KUKA KRL program: EPS_2_251503_MH01A_A_20251120020554.src

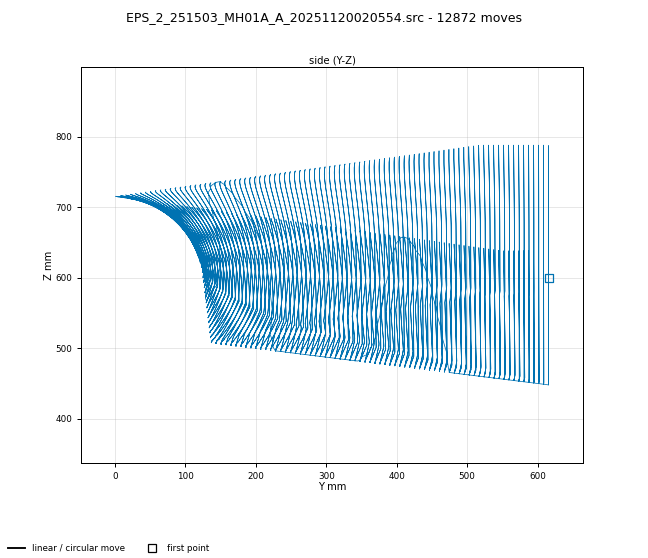
[picture p0: tool path of EPS_2_251503_MH01A_A_20251120020554.src, 12872 of 12874 moves have a stored position in this frame; points joined in program order, loops and branches not executed]
&ACCESS RVP
&REL 4
&COMMENT QRS 19112012
&PARAM EDITMASK = *
DEF PART()
EXT BAS (BAS_COMMAND :IN,REAL :IN )
INT I
BAS (#INITMOV,0 )

;KUKA QRS Post kuka4.cps  Date:22-06-2017 !

File_ID=2923

QRS_PRE_INIT()

;Init var - Until changes are made in qrs_pre_init
Outlet_Square_prg=0
Inlet_1_Square_prg=0
Inlet_2_Square_prg=0
Inlet_3_Square_prg=0
Inlet_4_Square_prg=0
Inlet_5_Square_prg=0

Outlet_1={X 0.000, Y 519.160, Z 687.500, B 0.000, E1 0.000 }
Inlet_1={X 0.000, Y 547.680, Z 287.500, B 0.000, E1 180.000 }
Outlet_1_type=201
Inlet_1_type=201
;QRS#1=Sidecore dimensions
;QRS#2=200-8" PVC SDR 35
;QRS#3=200-8" PVC SDR 35
;QRS#4=
;QRS#5=
;QRS#6=
;QRS#7=
;QRS#8=
;QRS#9=12-08 PSX
;QRS#10=12-08 PSX
;QRS#11=
;QRS#12=
;QRS#13=
;QRS#14=
;QRS#15=
;QRS#16=1220x127x1067 3,5'
;QRS#17=EPS Height
;QRS#18=788
;QRS#19=*
;QRS#20= UPDATED VERSION 22-06-2017
;QRS#21=*
Outlet_Square=0100
Inlet_1_Square=0100
Inlet_2_Square=0
Inlet_3_Square=0
Inlet_4_Square=0
Inlet_5_Square=0
Mill_Square=1
Outlet_Square_Prg=204
Inlet_1_Square_prg=204

QRS_INIT()

$ADVANCE=5

; T1
PTP {E1 173.592,E2 173.592}
PTP {X 0,Y 615.509,A -85,B 0,C 180,E1 173.592,E2 173.592,E3 0,E4 0,E5 0,E6 0}
QRS_SPEED_INIT()
LIN {X 0,Y 615.509,Z 600,A -85,B 0,C 180,E1 173.592,E2 173.592,E3 0,E4 0,E5 0,E6 0} C_VEL
LIN {X 0,Y 615.509,Z 457.87,A -85,B 0,C 180,E1 173.592,E2 173.592} C_VEL
LIN {X 0,Y 615.509,Z 449.7,A -85,B 0,C 180,E1 173.592,E2 173.592} C_VEL
LIN {X 0,Y 615.492,Z 447.7,A -85,B 0,C 180,E1 173.406,E2 173.406} C_VEL
LIN {X 0,Y 615.481,Z 447.688,A -85,B 0,C 180,E1 170.801,E2 170.801} C_VEL
LIN {X 0,Y 615.481,Z 447.684,A -85,B 0,C 180,E1 168.139,E2 168.139} C_VEL
LIN {X 0,Y 615.49,Z 447.696,A -85,B 0,C 180,E1 165.451,E2 165.451} C_VEL
LIN {X 0,Y 615.483,Z 447.687,A -85,B 0,C 180,E1 162.729,E2 162.729} C_VEL
LIN {X 0,Y 615.477,Z 447.685,A -85,B 0,C 180,E1 159.967,E2 159.967} C_VEL
LIN {X 0,Y 615.492,Z 447.699,A -85,B 0,C 180,E1 157.156,E2 157.156} C_VEL
LIN {X 0,Y 615.493,Z 447.68,A -85,B 0,C 180,E1 154.284,E2 154.284} C_VEL
LIN {X 0,Y 615.49,Z 447.696,A -85,B 0,C 180,E1 151.342,E2 151.342} C_VEL
LIN {X 0,Y 615.487,Z 447.694,A -85,B 0,C 180,E1 148.912,E2 148.912} C_VEL
LIN {X 0,Y 615.488,Z 447.684,A -85,B 0,C 180,E1 146.464,E2 146.464} C_VEL
LIN {X 0,Y 615.486,Z 447.682,A -85,B 0,C 180,E1 144.165,E2 144.165} C_VEL
LIN {X 0,Y 615.478,Z 447.684,A -85,B 0,C 180,E1 141.931,E2 141.931} C_VEL
LIN {X 0,Y 615.485,Z 447.692,A -85,B 0,C 180,E1 139.393,E2 139.393} C_VEL
LIN {X 0,Y 615.484,Z 447.693,A -85,B 0,C 180,E1 136.755,E2 136.755} C_VEL
LIN {X 0,Y 615.482,Z 447.683,A -85,B 0,C 180,E1 133.997,E2 133.997} C_VEL
LIN {X 0,Y 615.495,Z 447.698,A -85,B 0,C 180,E1 131.095,E2 131.095} C_VEL
LIN {X 0,Y 615.488,Z 447.681,A -85,B 0,C 180,E1 128.067,E2 128.067} C_VEL
LIN {X 0,Y 615.475,Z 447.687,A -85,B 0,C 180,E1 125.616,E2 125.616} C_VEL
LIN {X 0,Y 615.488,Z 447.692,A -85,B 0,C 180,E1 123.235,E2 123.235} C_VEL
LIN {X 0,Y 615.494,Z 447.701,A -85,B 0,C 180,E1 120.919,E2 120.919} C_VEL
LIN {X 0,Y 615.487,Z 447.688,A -85,B 0,C 180,E1 118.45,E2 118.45} C_VEL
LIN {X 0,Y 615.477,Z 447.684,A -85,B 0,C 180,E1 115.716,E2 115.716} C_VEL
LIN {X 0,Y 615.493,Z 447.701,A -85,B 0,C 180,E1 112.844,E2 112.844} C_VEL
LIN {X 0,Y 615.492,Z 447.681,A -85,B 0,C 180,E1 110.032,E2 110.032} C_VEL
LIN {X 0,Y 615.485,Z 447.688,A -85,B 0,C 180,E1 107.27,E2 107.27} C_VEL
LIN {X 0,Y 615.489,Z 447.693,A -85,B 0,C 180,E1 104.549,E2 104.549} C_VEL
LIN {X 0,Y 615.498,Z 447.906,A -85,B 0,C 180,E1 102.676,E2 102.676} C_VEL
LIN {X 0,Y 615.497,Z 448.814,A -85,B 0,C 180,E1 102.572,E2 102.572} C_VEL
LIN {X 0,Y 615.497,Z 534.805,A -85,B 0,C 180,E1 101.526,E2 101.526} C_VEL
LIN {X 0,Y 615.498,Z 547.747,A -85,B 0,C 180,E1 101.234,E2 101.234} C_VEL
LIN {X 0,Y 615.498,Z 560.738,A -85,B 0,C 180,E1 100.8,E2 100.8} C_VEL
LIN {X 0,Y 615.497,Z 572.199,A -85,B 0,C 180,E1 100.277,E2 100.277} C_VEL
LIN {X 0,Y 615.489,Z 583.581,A -85,B 0,C 180,E1 99.613,E2 99.613} C_VEL
LIN {X 0,Y 615.498,Z 593.825,A -85,B 0,C 180,E1 98.867,E2 98.867} C_VEL
LIN {X 0,Y 615.499,Z 603.036,A -85,B 0,C 180,E1 98.04,E2 98.04} C_VEL
LIN {X 0,Y 615.499,Z 611.893,A -85,B 0,C 180,E1 97.057,E2 97.057} C_VEL
LIN {X 0,Y 615.497,Z 619.124,A -85,B 0,C 180,E1 96.063,E2 96.063} C_VEL
LIN {X 0,Y 615.497,Z 623.959,A -85,B 0,C 180,E1 95.241,E2 95.241} C_VEL
LIN {X 0,Y 615.494,Z 628.658,A -85,B 0,C 180,E1 94.256,E2 94.256} C_VEL
LIN {X 0,Y 615.494,Z 632.255,A -85,B 0,C 180,E1 93.273,E2 93.273} C_VEL
LIN {X 0,Y 615.496,Z 634.115,A -85,B 0,C 180,E1 92.618,E2 92.618} C_VEL
LIN {X 0,Y 615.498,Z 635.533,A -85,B 0,C 180,E1 91.963,E2 91.963} C_VEL
LIN {X 0,Y 615.496,Z 637.142,A -85,B 0,C 180,E1 90.654,E2 90.654} C_VEL
LIN {X 0,Y 615.495,Z 637.384,A -85,B 0,C 180,E1 90,E2 90} C_VEL
LIN {X 0,Y 615.495,Z 637.206,A -85,B 0,C 180,E1 89.346,E2 89.346} C_VEL
LIN {X 0,Y 615.499,Z 635.682,A -85,B 0,C 180,E1 88.037,E2 88.037} C_VEL
LIN {X 0,Y 615.498,Z 634.341,A -85,B 0,C 180,E1 87.382,E2 87.382} C_VEL
LIN {X 0,Y 615.496,Z 631.494,A -85,B 0,C 180,E1 86.399,E2 86.399} C_VEL
LIN {X 0,Y 615.498,Z 627.635,A -85,B 0,C 180,E1 85.416,E2 85.416} C_VEL
LIN {X 0,Y 615.498,Z 622.652,A -85,B 0,C 180,E1 84.43,E2 84.43} C_VEL
LIN {X 0,Y 615.496,Z 616.208,A -85,B 0,C 180,E1 83.418,E2 83.418} C_VEL
LIN {X 0,Y 615.497,Z 608.538,A -85,B 0,C 180,E1 82.455,E2 82.455} C_VEL
LIN {X 0,Y 615.498,Z 598.761,A -85,B 0,C 180,E1 81.464,E2 81.464} C_VEL
LIN {X 0,Y 615.498,Z 588.496,A -85,B 0,C 180,E1 80.636,E2 80.636} C_VEL
LIN {X 0,Y 615.496,Z 576.933,A -85,B 0,C 180,E1 79.889,E2 79.889} C_VEL
LIN {X 0,Y 615.499,Z 565.025,A -85,B 0,C 180,E1 79.291,E2 79.291} C_VEL
LIN {X 0,Y 615.498,Z 552.166,A -85,B 0,C 180,E1 78.807,E2 78.807} C_VEL
LIN {X 0,Y 615.497,Z 539.569,A -85,B 0,C 180,E1 78.474,E2 78.474} C_VEL
LIN {X 0,Y 615.498,Z 526.457,A -85,B 0,C 180,E1 78.265,E2 78.265} C_VEL
LIN {X 0,Y 615.498,Z 448.939,A -85,B 0,C 180,E1 77.345,E2 77.345} C_VEL
LIN {X 0,Y 615.497,Z 447.856,A -85,B 0,C 180,E1 77.219,E2 77.219} C_VEL
LIN {X 0,Y 615.489,Z 447.691,A -85,B 0,C 180,E1 74.774,E2 74.774} C_VEL
LIN {X 0,Y 615.486,Z 447.682,A -85,B 0,C 180,E1 72.043,E2 72.043} C_VEL
LIN {X 0,Y 615.485,Z 447.696,A -85,B 0,C 180,E1 69.27,E2 69.27} C_VEL
LIN {X 0,Y 615.487,Z 447.699,A -85,B 0,C 180,E1 67.156,E2 67.156} C_VEL
LIN {X 0,Y 615.477,Z 447.687,A -85,B 0,C 180,E1 64.434,E2 64.434} C_VEL
LIN {X 0,Y 615.483,Z 447.683,A -85,B 0,C 180,E1 62.085,E2 62.085} C_VEL
LIN {X 0,Y 615.499,Z 447.679,A -85,B 0,C 180,E1 59.841,E2 59.841} C_VEL
LIN {X 0,Y 615.485,Z 447.686,A -85,B 0,C 180,E1 57.543,E2 57.543} C_VEL
LIN {X 0,Y 615.482,Z 447.696,A -85,B 0,C 180,E1 55.186,E2 55.186} C_VEL
LIN {X 0,Y 615.492,Z 447.694,A -85,B 0,C 180,E1 52.759,E2 52.759} C_VEL
LIN {X 0,Y 615.489,Z 447.681,A -85,B 0,C 180,E1 49.911,E2 49.911} C_VEL
LIN {X 0,Y 615.489,Z 447.701,A -85,B 0,C 180,E1 46.953,E2 46.953} C_VEL
LIN {X 0,Y 615.482,Z 447.683,A -85,B 0,C 180,E1 43.998,E2 43.998} C_VEL
LIN {X 0,Y 615.486,Z 447.694,A -85,B 0,C 180,E1 41.096,E2 41.096} C_VEL
LIN {X 0,Y 615.492,Z 447.7,A -85,B 0,C 180,E1 38.904,E2 38.904} C_VEL
LIN {X 0,Y 615.481,Z 447.691,A -85,B 0,C 180,E1 36.425,E2 36.425} C_VEL
LIN {X 0,Y 615.479,Z 447.684,A -85,B 0,C 180,E1 34.023,E2 34.023} C_VEL
LIN {X 0,Y 615.486,Z 447.682,A -85,B 0,C 180,E1 31.686,E2 31.686} C_VEL
LIN {X 0,Y 615.485,Z 447.685,A -85,B 0,C 180,E1 29.407,E2 29.407} C_VEL
LIN {X 0,Y 615.482,Z 447.694,A -85,B 0,C 180,E1 27.047,E2 27.047} C_VEL
LIN {X 0,Y 615.478,Z 447.69,A -85,B 0,C 180,E1 24.273,E2 24.273} C_VEL
LIN {X 0,Y 615.487,Z 447.683,A -85,B 0,C 180,E1 21.432,E2 21.432} C_VEL
LIN {X 0,Y 615.493,Z 447.698,A -85,B 0,C 180,E1 18.61,E2 18.61} C_VEL
LIN {X 0,Y 615.478,Z 447.685,A -85,B 0,C 180,E1 15.906,E2 15.906} C_VEL
LIN {X 0,Y 615.48,Z 447.687,A -85,B 0,C 180,E1 13.201,E2 13.201} C_VEL
LIN {X 0,Y 615.49,Z 447.698,A -85,B 0,C 180,E1 10.527,E2 10.527} C_VEL
LIN {X 0,Y 615.479,Z 447.685,A -85,B 0,C 180,E1 7.876,E2 7.876} C_VEL
LIN {X 0,Y 615.482,Z 447.685,A -85,B 0,C 180,E1 5.241,E2 5.241} C_VEL
LIN {X 0,Y 615.495,Z 447.699,A -85,B 0,C 180,E1 2.618,E2 2.618} C_VEL
LIN {X 0,Y 615.477,Z 447.688,A -85,B 0,C 180,E1 0,E2 0} C_VEL
LIN {X 0,Y 615.492,Z 447.681,A -85,B 0,C 180,E1 -2.618,E2 -2.618} C_VEL
LIN {X 0,Y 615.484,Z 447.695,A -85,B 0,C 180,E1 -5.241,E2 -5.241} C_VEL
LIN {X 0,Y 615.479,Z 447.692,A -85,B 0,C 180,E1 -7.876,E2 -7.876} C_VEL
LIN {X 0,Y 615.489,Z 447.681,A -85,B 0,C 180,E1 -10.527,E2 -10.527} C_VEL
LIN {X 0,Y 615.48,Z 447.693,A -85,B 0,C 180,E1 -13.201,E2 -13.201} C_VEL
LIN {X 0,Y 615.48,Z 447.693,A -85,B 0,C 180,E1 -15.905,E2 -15.905} C_VEL
LIN {X 0,Y 615.49,Z 447.681,A -85,B 0,C 180,E1 -18.646,E2 -18.646} C_VEL
LIN {X 0,Y 615.487,Z 447.696,A -85,B 0,C 180,E1 -21.432,E2 -21.432} C_VEL
LIN {X 0,Y 615.478,Z 447.686,A -85,B 0,C 180,E1 -24.272,E2 -24.272} C_VEL
LIN {X 0,Y 615.478,Z 447.687,A -85,B 0,C 180,E1 -27.046,E2 -27.046} C_VEL
LIN {X 0,Y 615.488,Z 447.698,A -85,B 0,C 180,E1 -29.797,E2 -29.797} C_VEL
LIN {X 0,Y 615.484,Z 447.683,A -85,B 0,C 180,E1 -32.458,E2 -32.458} C_VEL
LIN {X 0,Y 615.49,Z 447.681,A -85,B 0,C 180,E1 -34.815,E2 -34.815} C_VEL
LIN {X 0,Y 615.473,Z 447.69,A -85,B 0,C 180,E1 -37.243,E2 -37.243} C_VEL
LIN {X 0,Y 615.479,Z 447.693,A -85,B 0,C 180,E1 -40.09,E2 -40.09} C_VEL
LIN {X 0,Y 615.479,Z 447.687,A -85,B 0,C 180,E1 -42.354,E2 -42.354} C_VEL
LIN {X 0,Y 615.479,Z 447.685,A -85,B 0,C 180,E1 -45.07,E2 -45.07} C_VEL
LIN {X 0,Y 615.491,Z 447.698,A -85,B 0,C 180,E1 -47.92,E2 -47.92} C_VEL
LIN {X 0,Y 615.479,Z 447.69,A -85,B 0,C 180,E1 -50.25,E2 -50.25} C_VEL
LIN {X 0,Y 615.48,Z 447.684,A -85,B 0,C 180,E1 -53.065,E2 -53.065} C_VEL
LIN {X 0,Y 615.491,Z 447.698,A -85,B 0,C 180,E1 -55.979,E2 -55.979} C_VEL
LIN {X 0,Y 615.487,Z 447.682,A -85,B 0,C 180,E1 -58.914,E2 -58.914} C_VEL
LIN {X 0,Y 615.481,Z 447.692,A -85,B 0,C 180,E1 -61.551,E2 -61.551} C_VEL
LIN {X 0,Y 615.498,Z 447.813,A -85,B 0,C 180,E1 -64.013,E2 -64.013} C_VEL
LIN {X 0,Y 615.496,Z 448.16,A -85,B 0,C 180,E1 -64.104,E2 -64.104} C_VEL
LIN {X 0,Y 615.488,Z 473.307,A -85,B 0,C 180,E1 -66.801,E2 -66.801} C_VEL
LIN {X 0,Y 615.48,Z 499.798,A -85,B 0,C 180,E1 -69.577,E2 -69.577} C_VEL
LIN {X 0,Y 615.483,Z 527.091,A -85,B 0,C 180,E1 -72.387,E2 -72.387} C_VEL
LIN {X 0,Y 615.495,Z 553.944,A -85,B 0,C 180,E1 -75.113,E2 -75.113} C_VEL
LIN {X 0,Y 615.487,Z 573.871,A -85,B 0,C 180,E1 -77.093,E2 -77.093} C_VEL
LIN {X 0,Y 615.483,Z 683.847,A -85,B 0,C 180,E1 -78.411,E2 -78.411} C_VEL
LIN {X 0,Y 615.499,Z 696.352,A -85,B 0,C 180,E1 -78.682,E2 -78.682} C_VEL
LIN {X 0,Y 615.496,Z 709.5,A -85,B 0,C 180,E1 -79.109,E2 -79.109} C_VEL
LIN {X 0,Y 615.487,Z 721.482,A -85,B 0,C 180,E1 -79.64,E2 -79.64} C_VEL
LIN {X 0,Y 615.482,Z 733,A -85,B 0,C 180,E1 -80.304,E2 -80.304} C_VEL
LIN {X 0,Y 615.499,Z 743.344,A -85,B 0,C 180,E1 -81.05,E2 -81.05} C_VEL
LIN {X 0,Y 615.497,Z 751.814,A -85,B 0,C 180,E1 -81.794,E2 -81.794} C_VEL
LIN {X 0,Y 615.498,Z 759.608,A -85,B 0,C 180,E1 -82.62,E2 -82.62} C_VEL
LIN {X 0,Y 615.496,Z 767.204,A -85,B 0,C 180,E1 -83.608,E2 -83.608} C_VEL
LIN {X 0,Y 615.498,Z 774.205,A -85,B 0,C 180,E1 -84.759,E2 -84.759} C_VEL
LIN {X 0,Y 615.493,Z 778.852,A -85,B 0,C 180,E1 -85.744,E2 -85.744} C_VEL
LIN {X 0,Y 615.495,Z 782.399,A -85,B 0,C 180,E1 -86.727,E2 -86.727} C_VEL
LIN {X 0,Y 615.497,Z 784.233,A -85,B 0,C 180,E1 -87.382,E2 -87.382} C_VEL
LIN {X 0,Y 615.496,Z 785.608,A -85,B 0,C 180,E1 -88.037,E2 -88.037} C_VEL
LIN {X 0,Y 615.496,Z 787.174,A -85,B 0,C 180,E1 -89.346,E2 -89.346} C_VEL
LIN {X 0,Y 615.494,Z 787.389,A -85,B 0,C 180,E1 -90,E2 -90} C_VEL
LIN {X 0,Y 615.496,Z 786.58,A -85,B 0,C 180,E1 -91.309,E2 -91.309} C_VEL
LIN {X 0,Y 615.496,Z 785.608,A -85,B 0,C 180,E1 -91.963,E2 -91.963} C_VEL
LIN {X 0,Y 615.497,Z 784.233,A -85,B 0,C 180,E1 -92.618,E2 -92.618} C_VEL
LIN {X 0,Y 615.496,Z 781.35,A -85,B 0,C 180,E1 -93.601,E2 -93.601} C_VEL
LIN {X 0,Y 615.498,Z 777.442,A -85,B 0,C 180,E1 -94.584,E2 -94.584} C_VEL
LIN {X 0,Y 615.499,Z 772.406,A -85,B 0,C 180,E1 -95.57,E2 -95.57} C_VEL
LIN {X 0,Y 615.497,Z 765.869,A -85,B 0,C 180,E1 -96.583,E2 -96.583} C_VEL
LIN {X 0,Y 615.497,Z 758.135,A -85,B 0,C 180,E1 -97.545,E2 -97.545} C_VEL
LIN {X 0,Y 615.498,Z 750.047,A -85,B 0,C 180,E1 -98.371,E2 -98.371} C_VEL
LIN {X 0,Y 615.499,Z 740.17,A -85,B 0,C 180,E1 -99.198,E2 -99.198} C_VEL
LIN {X 0,Y 615.483,Z 728.986,A -85,B 0,C 180,E1 -99.945,E2 -99.945} C_VEL
LIN {X 0,Y 615.489,Z 718.027,A -85,B 0,C 180,E1 -100.527,E2 -100.527} C_VEL
LIN {X 0,Y 615.499,Z 705.418,A -85,B 0,C 180,E1 -101.042,E2 -101.042} C_VEL
LIN {X 0,Y 615.497,Z 693.075,A -85,B 0,C 180,E1 -101.401,E2 -101.401} C_VEL
LIN {X 0,Y 615.479,Z 679.489,A -85,B 0,C 180,E1 -101.652,E2 -101.652} C_VEL
LIN {X 0,Y 615.487,Z 573.871,A -85,B 0,C 180,E1 -102.907,E2 -102.907} C_VEL
LIN {X 0,Y 615.48,Z 548.911,A -85,B 0,C 180,E1 -105.395,E2 -105.395} C_VEL
LIN {X 0,Y 615.489,Z 522.161,A -85,B 0,C 180,E1 -108.117,E2 -108.117} C_VEL
LIN {X 0,Y 615.484,Z 495.16,A -85,B 0,C 180,E1 -110.905,E2 -110.905} C_VEL
LIN {X 0,Y 615.477,Z 468.881,A -85,B 0,C 180,E1 -113.669,E2 -113.669} C_VEL
LIN {X 0,Y 615.495,Z 448.029,A -85,B 0,C 180,E1 -115.919,E2 -115.919} C_VEL
LIN {X 0,Y 615.498,Z 447.721,A -85,B 0,C 180,E1 -116.078,E2 -116.078} C_VEL
LIN {X 0,Y 615.477,Z 447.688,A -85,B 0,C 180,E1 -118.658,E2 -118.658} C_VEL
LIN {X 0,Y 615.487,Z 447.681,A -85,B 0,C 180,E1 -121.086,E2 -121.086} C_VEL
LIN {X 0,Y 615.491,Z 447.697,A -85,B 0,C 180,E1 -124.021,E2 -124.021} C_VEL
LIN {X 0,Y 615.48,Z 447.684,A -85,B 0,C 180,E1 -126.935,E2 -126.935} C_VEL
LIN {X 0,Y 615.478,Z 447.69,A -85,B 0,C 180,E1 -129.75,E2 -129.75} C_VEL
LIN {X 0,Y 615.49,Z 447.697,A -85,B 0,C 180,E1 -132.351,E2 -132.351} C_VEL
LIN {X 0,Y 615.48,Z 447.684,A -85,B 0,C 180,E1 -135.068,E2 -135.068} C_VEL
LIN {X 0,Y 615.477,Z 447.693,A -85,B 0,C 180,E1 -137.919,E2 -137.919} C_VEL
LIN {X 0,Y 615.498,Z 447.7,A -85,B 0,C 180,E1 -140.251,E2 -140.251} C_VEL
LIN {X 0,Y 615.478,Z 447.685,A -85,B 0,C 180,E1 -143.063,E2 -143.063} C_VEL
LIN {X 0,Y 615.49,Z 447.681,A -85,B 0,C 180,E1 -145.297,E2 -145.297} C_VEL
LIN {X 0,Y 615.479,Z 447.686,A -85,B 0,C 180,E1 -147.668,E2 -147.668} C_VEL
LIN {X 0,Y 615.488,Z 447.697,A -85,B 0,C 180,E1 -150.203,E2 -150.203} C_VEL
LIN {X 0,Y 615.478,Z 447.687,A -85,B 0,C 180,E1 -152.954,E2 -152.954} C_VEL
LIN {X 0,Y 615.478,Z 447.686,A -85,B 0,C 180,E1 -155.728,E2 -155.728} C_VEL
LIN {X 0,Y 615.489,Z 447.697,A -85,B 0,C 180,E1 -158.568,E2 -158.568} C_VEL
LIN {X 0,Y 615.492,Z 447.68,A -85,B 0,C 180,E1 -161.39,E2 -161.39} C_VEL
LIN {X 0,Y 615.48,Z 447.692,A -85,B 0,C 180,E1 -164.095,E2 -164.095} C_VEL
LIN {X 0,Y 615.48,Z 447.693,A -85,B 0,C 180,E1 -166.799,E2 -166.799} C_VEL
LIN {X 0,Y 615.489,Z 447.681,A -85,B 0,C 180,E1 -169.473,E2 -169.473} C_VEL
LIN {X 0,Y 615.477,Z 447.691,A -85,B 0,C 180,E1 -172.124,E2 -172.124} C_VEL
LIN {X 0,Y 615.486,Z 447.695,A -85,B 0,C 180,E1 -174.759,E2 -174.759} C_VEL
LIN {X 0,Y 615.492,Z 447.681,A -85,B 0,C 180,E1 -177.382,E2 -177.382} C_VEL
LIN {X 0,Y 615.477,Z 447.687,A -85,B 0,C 180,E1 -180,E2 -180} C_VEL
LIN {X 0,Y 615.495,Z 447.701,A -85,B 0,C 180,E1 -182.618,E2 -182.618} C_VEL
LIN {X 0,Y 615.48,Z 447.687,A -85,B 0,C 180,E1 -185.241,E2 -185.241} C_VEL
LIN {X 0,Y 615.492,Z 447.7,A -85,B 0,C 180,E1 -186.594,E2 -186.594} C_VEL
LIN {X 0,Y 614.81,Z 447.835,A -85,B 0,C 180,E1 -187.14,E2 -187.14} C_VEL
LIN {X 0,Y 611.97,Z 448.25,A -85,B 0,C 180,E1 -188.026,E2 -188.026} C_VEL
LIN {X 0,Y 609.576,Z 448.56,A -85,B 0,C 180,E1 -188.738,E2 -188.738} C_VEL
LIN {X 0,Y 608.541,Z 448.678,A -85,B 0,C 180,E1 -189.288,E2 -189.288} C_VEL
LIN {X 0,Y 608.453,Z 448.687,A -85,B 0,C 180,E1 -189.474,E2 -189.474} C_VEL
LIN {X 0,Y 608.457,Z 448.687,A -85,B 0,C 180,E1 -192,E2 -192} C_VEL
LIN {X 0,Y 608.475,Z 448.695,A -85,B 0,C 180,E1 -194.721,E2 -194.721} C_VEL
LIN {X 0,Y 608.448,Z 448.688,A -85,B 0,C 180,E1 -197.477,E2 -197.477} C_VEL
LIN {X 0,Y 608.459,Z 448.689,A -85,B 0,C 180,E1 -200.274,E2 -200.274} C_VEL
LIN {X 0,Y 608.453,Z 448.692,A -85,B 0,C 180,E1 -203.124,E2 -203.124} C_VEL
LIN {X 0,Y 608.447,Z 448.688,A -85,B 0,C 180,E1 -206.036,E2 -206.036} C_VEL
LIN {X 0,Y 608.471,Z 448.692,A -85,B 0,C 180,E1 -208.622,E2 -208.622} C_VEL
LIN {X 0,Y 608.472,Z 448.687,A -85,B 0,C 180,E1 -211.316,E2 -211.316} C_VEL
LIN {X 0,Y 608.471,Z 448.685,A -85,B 0,C 180,E1 -213.737,E2 -213.737} C_VEL
LIN {X 0,Y 608.472,Z 448.685,A -85,B 0,C 180,E1 -216.091,E2 -216.091} C_VEL
LIN {X 0,Y 608.471,Z 448.69,A -85,B 0,C 180,E1 -218.588,E2 -218.588} C_VEL
LIN {X 0,Y 608.463,Z 448.689,A -85,B 0,C 180,E1 -221.344,E2 -221.344} C_VEL
LIN {X 0,Y 608.449,Z 448.688,A -85,B 0,C 180,E1 -224.265,E2 -224.265} C_VEL
LIN {X 0,Y 608.46,Z 448.696,A -85,B 0,C 180,E1 -227.042,E2 -227.042} C_VEL
LIN {X 0,Y 608.454,Z 448.688,A -85,B 0,C 180,E1 -229.698,E2 -229.698} C_VEL
LIN {X 0,Y 608.47,Z 448.685,A -85,B 0,C 180,E1 -232.255,E2 -232.255} C_VEL
LIN {X 0,Y 608.481,Z 448.693,A -85,B 0,C 180,E1 -235.091,E2 -235.091} C_VEL
LIN {X 0,Y 608.467,Z 448.685,A -85,B 0,C 180,E1 -237.906,E2 -237.906} C_VEL
LIN {X 0,Y 608.461,Z 448.686,A -85,B 0,C 180,E1 -240.221,E2 -240.221} C_VEL
LIN {X 0,Y 608.484,Z 448.688,A -85,B 0,C 180,E1 -242.792,E2 -242.792} C_VEL
LIN {X 0,Y 608.483,Z 448.684,A -85,B 0,C 180,E1 -245.847,E2 -245.847} C_VEL
LIN {X 0,Y 608.468,Z 448.685,A -85,B 0,C 180,E1 -248.309,E2 -248.309} C_VEL
LIN {X 0,Y 608.457,Z 448.697,A -85,B 0,C 180,E1 -251.131,E2 -251.131} C_VEL
LIN {X 0,Y 608.462,Z 448.687,A -85,B 0,C 180,E1 -253.907,E2 -253.907} C_VEL
LIN {X 0,Y 608.465,Z 448.688,A -85,B 0,C 180,E1 -256.644,E2 -256.644} C_VEL
LIN {X 0,Y 608.509,Z 448.94,A -85,B 0,C 180,E1 -257.218,E2 -257.218} C_VEL
LIN {X 0,Y 608.589,Z 449.922,A -85,B 0,C 180,E1 -257.305,E2 -257.305} C_VEL
LIN {X 0,Y 608.558,Z 533.811,A -85,B 0,C 180,E1 -258.319,E2 -258.319} C_VEL
LIN {X 0,Y 608.538,Z 547.126,A -85,B 0,C 180,E1 -258.614,E2 -258.614} C_VEL
LIN {X 0,Y 608.529,Z 560.355,A -85,B 0,C 180,E1 -259.055,E2 -259.055} C_VEL
LIN {X 0,Y 608.508,Z 572.374,A -85,B 0,C 180,E1 -259.604,E2 -259.604} C_VEL
LIN {X 0,Y 608.5,Z 583.794,A -85,B 0,C 180,E1 -260.276,E2 -260.276} C_VEL
LIN {X 0,Y 608.474,Z 594.087,A -85,B 0,C 180,E1 -261.03,E2 -261.03} C_VEL
LIN {X 0,Y 608.464,Z 603.352,A -85,B 0,C 180,E1 -261.866,E2 -261.866} C_VEL
LIN {X 0,Y 608.466,Z 612.325,A -85,B 0,C 180,E1 -262.868,E2 -262.868} C_VEL
LIN {X 0,Y 608.444,Z 619.556,A -85,B 0,C 180,E1 -263.867,E2 -263.867} C_VEL
LIN {X 0,Y 608.462,Z 624.435,A -85,B 0,C 180,E1 -264.698,E2 -264.698} C_VEL
LIN {X 0,Y 608.439,Z 629.179,A -85,B 0,C 180,E1 -265.694,E2 -265.694} C_VEL
LIN {X 0,Y 608.425,Z 632.812,A -85,B 0,C 180,E1 -266.689,E2 -266.689} C_VEL
LIN {X 0,Y 608.425,Z 634.691,A -85,B 0,C 180,E1 -267.352,E2 -267.352} C_VEL
LIN {X 0,Y 608.443,Z 636.127,A -85,B 0,C 180,E1 -268.014,E2 -268.014} C_VEL
LIN {X 0,Y 608.439,Z 637.752,A -85,B 0,C 180,E1 -269.338,E2 -269.338} C_VEL
LIN {X 0,Y 608.435,Z 637.995,A -85,B 0,C 180,E1 -270,E2 -270} C_VEL
LIN {X 0,Y 608.438,Z 637.815,A -85,B 0,C 180,E1 -270.662,E2 -270.662} C_VEL
LIN {X 0,Y 608.444,Z 636.276,A -85,B 0,C 180,E1 -271.986,E2 -271.986} C_VEL
LIN {X 0,Y 608.426,Z 634.919,A -85,B 0,C 180,E1 -272.648,E2 -272.648} C_VEL
LIN {X 0,Y 608.449,Z 632.042,A -85,B 0,C 180,E1 -273.642,E2 -273.642} C_VEL
LIN {X 0,Y 608.433,Z 628.143,A -85,B 0,C 180,E1 -274.638,E2 -274.638} C_VEL
LIN {X 0,Y 608.449,Z 623.113,A -85,B 0,C 180,E1 -275.634,E2 -275.634} C_VEL
LIN {X 0,Y 608.441,Z 616.796,A -85,B 0,C 180,E1 -276.633,E2 -276.633} C_VEL
LIN {X 0,Y 608.475,Z 608.88,A -85,B 0,C 180,E1 -277.633,E2 -277.633} C_VEL
LIN {X 0,Y 608.472,Z 599.038,A -85,B 0,C 180,E1 -278.636,E2 -278.636} C_VEL
LIN {X 0,Y 608.479,Z 588.717,A -85,B 0,C 180,E1 -279.473,E2 -279.473} C_VEL
LIN {X 0,Y 608.493,Z 577.104,A -85,B 0,C 180,E1 -280.229,E2 -280.229} C_VEL
LIN {X 0,Y 608.529,Z 565.859,A -85,B 0,C 180,E1 -280.803,E2 -280.803} C_VEL
LIN {X 0,Y 608.538,Z 554.268,A -85,B 0,C 180,E1 -281.257,E2 -281.257} C_VEL
LIN {X 0,Y 608.539,Z 540.573,A -85,B 0,C 180,E1 -281.639,E2 -281.639} C_VEL
LIN {X 0,Y 608.573,Z 528.311,A -85,B 0,C 180,E1 -281.849,E2 -281.849} C_VEL
LIN {X 0,Y 608.593,Z 450.076,A -85,B 0,C 180,E1 -282.78,E2 -282.78} C_VEL
LIN {X 0,Y 608.51,Z 448.862,A -85,B 0,C 180,E1 -282.888,E2 -282.888} C_VEL
LIN {X 0,Y 608.473,Z 448.687,A -85,B 0,C 180,E1 -285.405,E2 -285.405} C_VEL
LIN {X 0,Y 608.449,Z 448.687,A -85,B 0,C 180,E1 -288.171,E2 -288.171} C_VEL
LIN {X 0,Y 608.455,Z 448.697,A -85,B 0,C 180,E1 -290.981,E2 -290.981} C_VEL
LIN {X 0,Y 608.447,Z 448.695,A -85,B 0,C 180,E1 -293.124,E2 -293.124} C_VEL
LIN {X 0,Y 608.464,Z 448.686,A -85,B 0,C 180,E1 -295.719,E2 -295.719} C_VEL
LIN {X 0,Y 608.45,Z 448.688,A -85,B 0,C 180,E1 -298.266,E2 -298.266} C_VEL
LIN {X 0,Y 608.478,Z 448.687,A -85,B 0,C 180,E1 -300.544,E2 -300.544} C_VEL
LIN {X 0,Y 608.458,Z 448.695,A -85,B 0,C 180,E1 -302.879,E2 -302.879} C_VEL
LIN {X 0,Y 608.436,Z 448.695,A -85,B 0,C 180,E1 -305.277,E2 -305.277} C_VEL
LIN {X 0,Y 608.47,Z 448.686,A -85,B 0,C 180,E1 -307.745,E2 -307.745} C_VEL
LIN {X 0,Y 608.452,Z 448.688,A -85,B 0,C 180,E1 -310.329,E2 -310.329} C_VEL
LIN {X 0,Y 608.484,Z 448.69,A -85,B 0,C 180,E1 -313.31,E2 -313.31} C_VEL
LIN {X 0,Y 608.467,Z 448.685,A -85,B 0,C 180,E1 -316.13,E2 -316.13} C_VEL
LIN {X 0,Y 608.455,Z 448.692,A -85,B 0,C 180,E1 -318.823,E2 -318.823} C_VEL
LIN {X 0,Y 608.469,Z 448.691,A -85,B 0,C 180,E1 -321.412,E2 -321.412} C_VEL
LIN {X 0,Y 608.471,Z 448.685,A -85,B 0,C 180,E1 -323.949,E2 -323.949} C_VEL
LIN {X 0,Y 608.462,Z 448.686,A -85,B 0,C 180,E1 -326.329,E2 -326.329} C_VEL
LIN {X 0,Y 608.472,Z 448.687,A -85,B 0,C 180,E1 -328.726,E2 -328.726} C_VEL
LIN {X 0,Y 608.474,Z 448.692,A -85,B 0,C 180,E1 -331.377,E2 -331.377} C_VEL
LIN {X 0,Y 608.475,Z 448.684,A -85,B 0,C 180,E1 -334.276,E2 -334.276} C_VEL
LIN {X 0,Y 608.452,Z 448.691,A -85,B 0,C 180,E1 -336.876,E2 -336.876} C_VEL
LIN {X 0,Y 608.459,Z 448.69,A -85,B 0,C 180,E1 -339.726,E2 -339.726} C_VEL
LIN {X 0,Y 608.446,Z 448.688,A -85,B 0,C 180,E1 -342.523,E2 -342.523} C_VEL
LIN {X 0,Y 608.474,Z 448.694,A -85,B 0,C 180,E1 -345.279,E2 -345.279} C_VEL
LIN {X 0,Y 608.456,Z 448.688,A -85,B 0,C 180,E1 -348,E2 -348} C_VEL
LIN {X 0,Y 608.464,Z 448.686,A -85,B 0,C 180,E1 -350.694,E2 -350.694} C_VEL
LIN {X 0,Y 608.466,Z 448.696,A -85,B 0,C 180,E1 -353.367,E2 -353.367} C_VEL
LIN {X 0,Y 608.446,Z 448.689,A -85,B 0,C 180,E1 -356.026,E2 -356.026} C_VEL
LIN {X 0,Y 608.469,Z 448.685,A -85,B 0,C 180,E1 -358.676,E2 -358.676} C_VEL
LIN {X 0,Y 608.471,Z 448.693,A -85,B 0,C 180,E1 -361.324,E2 -361.324} C_VEL
LIN {X 0,Y 608.445,Z 448.69,A -85,B 0,C 180,E1 -363.974,E2 -363.974} C_VEL
LIN {X 0,Y 608.465,Z 448.685,A -85,B 0,C 180,E1 -366.633,E2 -366.633} C_VEL
LIN {X 0,Y 608.463,Z 448.693,A -85,B 0,C 180,E1 -369.306,E2 -369.306} C_VEL
LIN {X 0,Y 608.456,Z 448.69,A -85,B 0,C 180,E1 -372,E2 -372} C_VEL
LIN {X 0,Y 608.473,Z 448.685,A -85,B 0,C 180,E1 -374.721,E2 -374.721} C_VEL
LIN {X 0,Y 608.445,Z 448.697,A -85,B 0,C 180,E1 -377.477,E2 -377.477} C_VEL
LIN {X 0,Y 608.458,Z 448.687,A -85,B 0,C 180,E1 -380.274,E2 -380.274} C_VEL
LIN {X 0,Y 608.449,Z 448.687,A -85,B 0,C 180,E1 -382.477,E2 -382.477} C_VEL
LIN {X 0,Y 608.45,Z 448.692,A -85,B 0,C 180,E1 -385.301,E2 -385.301} C_VEL
LIN {X 0,Y 608.443,Z 448.697,A -85,B 0,C 180,E1 -387.518,E2 -387.518} C_VEL
LIN {X 0,Y 608.464,Z 448.691,A -85,B 0,C 180,E1 -389.973,E2 -389.973} C_VEL
LIN {X 0,Y 608.458,Z 448.686,A -85,B 0,C 180,E1 -392.524,E2 -392.524} C_VEL
LIN {X 0,Y 608.449,Z 448.691,A -85,B 0,C 180,E1 -395.277,E2 -395.277} C_VEL
LIN {X 0,Y 608.461,Z 448.688,A -85,B 0,C 180,E1 -398.241,E2 -398.241} C_VEL
LIN {X 0,Y 608.446,Z 448.69,A -85,B 0,C 180,E1 -400.33,E2 -400.33} C_VEL
LIN {X 0,Y 608.446,Z 448.688,A -85,B 0,C 180,E1 -402.961,E2 -402.961} C_VEL
LIN {X 0,Y 608.461,Z 448.696,A -85,B 0,C 180,E1 -405.736,E2 -405.736} C_VEL
LIN {X 0,Y 608.46,Z 448.686,A -85,B 0,C 180,E1 -408.658,E2 -408.658} C_VEL
LIN {X 0,Y 608.466,Z 448.689,A -85,B 0,C 180,E1 -411.413,E2 -411.413} C_VEL
LIN {X 0,Y 608.444,Z 448.697,A -85,B 0,C 180,E1 -413.955,E2 -413.955} C_VEL
LIN {X 0,Y 608.462,Z 448.689,A -85,B 0,C 180,E1 -416.33,E2 -416.33} C_VEL
LIN {X 0,Y 608.477,Z 448.684,A -85,B 0,C 180,E1 -418.728,E2 -418.728} C_VEL
LIN {X 0,Y 608.467,Z 448.688,A -85,B 0,C 180,E1 -421.382,E2 -421.382} C_VEL
LIN {X 0,Y 608.49,Z 448.884,A -85,B 0,C 180,E1 -423.852,E2 -423.852} C_VEL
LIN {X 0,Y 608.75,Z 452.023,A -85,B 0,C 180,E1 -424.225,E2 -424.225} C_VEL
LIN {X 0,Y 608.663,Z 476.669,A -85,B 0,C 180,E1 -426.885,E2 -426.885} C_VEL
LIN {X 0,Y 608.607,Z 503.565,A -85,B 0,C 180,E1 -429.731,E2 -429.731} C_VEL
LIN {X 0,Y 608.547,Z 530.46,A -85,B 0,C 180,E1 -432.527,E2 -432.527} C_VEL
LIN {X 0,Y 608.523,Z 555.675,A -85,B 0,C 180,E1 -435.11,E2 -435.11} C_VEL
LIN {X 0,Y 608.53,Z 573.91,A -85,B 0,C 180,E1 -436.943,E2 -436.943} C_VEL
LIN {X 0,Y 608.534,Z 683.962,A -85,B 0,C 180,E1 -438.277,E2 -438.277} C_VEL
LIN {X 0,Y 608.544,Z 697.226,A -85,B 0,C 180,E1 -438.572,E2 -438.572} C_VEL
LIN {X 0,Y 608.544,Z 710.333,A -85,B 0,C 180,E1 -439.009,E2 -439.009} C_VEL
LIN {X 0,Y 608.506,Z 721.64,A -85,B 0,C 180,E1 -439.519,E2 -439.519} C_VEL
LIN {X 0,Y 608.472,Z 733.201,A -85,B 0,C 180,E1 -440.191,E2 -440.191} C_VEL
LIN {X 0,Y 608.485,Z 743.596,A -85,B 0,C 180,E1 -440.946,E2 -440.946} C_VEL
LIN {X 0,Y 608.475,Z 752.114,A -85,B 0,C 180,E1 -441.699,E2 -441.699} C_VEL
LIN {X 0,Y 608.471,Z 759.962,A -85,B 0,C 180,E1 -442.534,E2 -442.534} C_VEL
LIN {X 0,Y 608.461,Z 767.287,A -85,B 0,C 180,E1 -443.485,E2 -443.485} C_VEL
LIN {X 0,Y 608.45,Z 772.867,A -85,B 0,C 180,E1 -444.366,E2 -444.366} C_VEL
LIN {X 0,Y 608.432,Z 777.951,A -85,B 0,C 180,E1 -445.362,E2 -445.362} C_VEL
LIN {X 0,Y 608.449,Z 781.896,A -85,B 0,C 180,E1 -446.358,E2 -446.358} C_VEL
LIN {X 0,Y 608.425,Z 784.809,A -85,B 0,C 180,E1 -447.352,E2 -447.352} C_VEL
LIN {X 0,Y 608.441,Z 786.201,A -85,B 0,C 180,E1 -448.014,E2 -448.014} C_VEL
LIN {X 0,Y 608.438,Z 787.783,A -85,B 0,C 180,E1 -449.338,E2 -449.338} C_VEL
LIN {X 0,Y 608.434,Z 788,A -85,B 0,C 180,E1 -450,E2 -450} C_VEL
LIN {X 0,Y 608.448,Z 787.184,A -85,B 0,C 180,E1 -451.324,E2 -451.324} C_VEL
LIN {X 0,Y 608.441,Z 786.201,A -85,B 0,C 180,E1 -451.986,E2 -451.986} C_VEL
LIN {X 0,Y 608.425,Z 784.809,A -85,B 0,C 180,E1 -452.648,E2 -452.648} C_VEL
LIN {X 0,Y 608.449,Z 781.896,A -85,B 0,C 180,E1 -453.642,E2 -453.642} C_VEL
LIN {X 0,Y 608.432,Z 777.951,A -85,B 0,C 180,E1 -454.638,E2 -454.638} C_VEL
LIN {X 0,Y 608.437,Z 771.877,A -85,B 0,C 180,E1 -455.801,E2 -455.801} C_VEL
LIN {X 0,Y 608.462,Z 765.236,A -85,B 0,C 180,E1 -456.799,E2 -456.799} C_VEL
LIN {X 0,Y 608.455,Z 756.991,A -85,B 0,C 180,E1 -457.8,E2 -457.8} C_VEL
LIN {X 0,Y 608.472,Z 748.539,A -85,B 0,C 180,E1 -458.636,E2 -458.636} C_VEL
LIN {X 0,Y 608.474,Z 738.094,A -85,B 0,C 180,E1 -459.473,E2 -459.473} C_VEL
LIN {X 0,Y 608.482,Z 727.76,A -85,B 0,C 180,E1 -460.145,E2 -460.145} C_VEL
LIN {X 0,Y 608.522,Z 716.243,A -85,B 0,C 180,E1 -460.741,E2 -460.741} C_VEL
LIN {X 0,Y 608.533,Z 704.879,A -85,B 0,C 180,E1 -461.192,E2 -461.192} C_VEL
LIN {X 0,Y 608.551,Z 691.365,A -85,B 0,C 180,E1 -461.575,E2 -461.575} C_VEL
LIN {X 0,Y 608.544,Z 678.106,A -85,B 0,C 180,E1 -461.808,E2 -461.808} C_VEL
LIN {X 0,Y 608.53,Z 573.909,A -85,B 0,C 180,E1 -463.057,E2 -463.057} C_VEL
LIN {X 0,Y 608.528,Z 545.589,A -85,B 0,C 180,E1 -465.919,E2 -465.919} C_VEL
LIN {X 0,Y 608.566,Z 519.442,A -85,B 0,C 180,E1 -468.613,E2 -468.613} C_VEL
LIN {X 0,Y 608.632,Z 493.479,A -85,B 0,C 180,E1 -471.329,E2 -471.329} C_VEL
LIN {X 0,Y 608.68,Z 467.807,A -85,B 0,C 180,E1 -474.066,E2 -474.066} C_VEL
LIN {X 0,Y 608.682,Z 449.774,A -85,B 0,C 180,E1 -476.024,E2 -476.024} C_VEL
LIN {X 0,Y 608.481,Z 448.744,A -85,B 0,C 180,E1 -476.194,E2 -476.194} C_VEL
LIN {X 0,Y 608.465,Z 448.686,A -85,B 0,C 180,E1 -479.019,E2 -479.019} C_VEL
LIN {X 0,Y 608.475,Z 448.684,A -85,B 0,C 180,E1 -481.315,E2 -481.315} C_VEL
LIN {X 0,Y 608.47,Z 448.689,A -85,B 0,C 180,E1 -483.734,E2 -483.734} C_VEL
LIN {X 0,Y 608.443,Z 448.698,A -85,B 0,C 180,E1 -486.091,E2 -486.091} C_VEL
LIN {X 0,Y 608.466,Z 448.689,A -85,B 0,C 180,E1 -488.587,E2 -488.587} C_VEL
LIN {X 0,Y 608.459,Z 448.686,A -85,B 0,C 180,E1 -491.342,E2 -491.342} C_VEL
LIN {X 0,Y 608.46,Z 448.696,A -85,B 0,C 180,E1 -494.264,E2 -494.264} C_VEL
LIN {X 0,Y 608.446,Z 448.688,A -85,B 0,C 180,E1 -497.039,E2 -497.039} C_VEL
LIN {X 0,Y 608.446,Z 448.69,A -85,B 0,C 180,E1 -499.696,E2 -499.696} C_VEL
LIN {X 0,Y 608.462,Z 448.696,A -85,B 0,C 180,E1 -502.253,E2 -502.253} C_VEL
LIN {X 0,Y 608.48,Z 448.684,A -85,B 0,C 180,E1 -505.088,E2 -505.088} C_VEL
LIN {X 0,Y 608.462,Z 448.689,A -85,B 0,C 180,E1 -507.905,E2 -507.905} C_VEL
LIN {X 0,Y 608.472,Z 448.693,A -85,B 0,C 180,E1 -510.221,E2 -510.221} C_VEL
LIN {X 0,Y 608.471,Z 448.688,A -85,B 0,C 180,E1 -512.791,E2 -512.791} C_VEL
LIN {X 0,Y 608.446,Z 448.688,A -85,B 0,C 180,E1 -515.429,E2 -515.429} C_VEL
LIN {X 0,Y 608.466,Z 448.694,A -85,B 0,C 180,E1 -518.308,E2 -518.308} C_VEL
LIN {X 0,Y 608.469,Z 448.685,A -85,B 0,C 180,E1 -521.281,E2 -521.281} C_VEL
LIN {X 0,Y 608.456,Z 448.689,A -85,B 0,C 180,E1 -523.906,E2 -523.906} C_VEL
LIN {X 0,Y 608.457,Z 448.694,A -85,B 0,C 180,E1 -526.643,E2 -526.643} C_VEL
LIN {X 0,Y 608.464,Z 448.685,A -85,B 0,C 180,E1 -529.35,E2 -529.35} C_VEL
LIN {X 0,Y 608.47,Z 448.688,A -85,B 0,C 180,E1 -532.033,E2 -532.033} C_VEL
LIN {X 0,Y 608.464,Z 448.694,A -85,B 0,C 180,E1 -534.698,E2 -534.698} C_VEL
LIN {X 0,Y 608.481,Z 448.684,A -85,B 0,C 180,E1 -537.352,E2 -537.352} C_VEL
LIN {X 0,Y 608.467,Z 448.687,A -85,B 0,C 180,E1 -540,E2 -540} C_VEL
LIN {X 0,Y 608.484,Z 448.694,A -85,B 0,C 180,E1 -542.648,E2 -542.648} C_VEL
LIN {X 0,Y 608.458,Z 448.687,A -85,B 0,C 180,E1 -545.302,E2 -545.302} C_VEL
LIN {X 0,Y 608.472,Z 448.685,A -85,B 0,C 180,E1 -547.967,E2 -547.967} C_VEL
LIN {X 0,Y 608.453,Z 448.687,A -85,B 0,C 180,E1 -549.474,E2 -549.474} C_VEL
LIN {X 0,Y 607.774,Z 448.773,A -85,B 0,C 180,E1 -550.027,E2 -550.027} C_VEL
LIN {X 0,Y 604.919,Z 449.134,A -85,B 0,C 180,E1 -550.924,E2 -550.924} C_VEL
LIN {X 0,Y 602.517,Z 449.43,A -85,B 0,C 180,E1 -551.645,E2 -551.645} C_VEL
LIN {X 0,Y 601.489,Z 449.557,A -85,B 0,C 180,E1 -552.202,E2 -552.202} C_VEL
LIN {X 0,Y 601.406,Z 449.568,A -85,B 0,C 180,E1 -552.39,E2 -552.39} C_VEL
LIN {X 0,Y 601.427,Z 449.569,A -85,B 0,C 180,E1 -554.897,E2 -554.897} C_VEL
LIN {X 0,Y 601.428,Z 449.568,A -85,B 0,C 180,E1 -556.986,E2 -556.986} C_VEL
LIN {X 0,Y 601.402,Z 449.565,A -85,B 0,C 180,E1 -559.81,E2 -559.81} C_VEL
LIN {X 0,Y 601.407,Z 449.572,A -85,B 0,C 180,E1 -562.607,E2 -562.607} C_VEL
LIN {X 0,Y 601.401,Z 449.575,A -85,B 0,C 180,E1 -564.879,E2 -564.879} C_VEL
LIN {X 0,Y 601.416,Z 449.563,A -85,B 0,C 180,E1 -567.868,E2 -567.868} C_VEL
LIN {X 0,Y 601.441,Z 449.56,A -85,B 0,C 180,E1 -570.164,E2 -570.164} C_VEL
LIN {X 0,Y 601.419,Z 449.57,A -85,B 0,C 180,E1 -572.717,E2 -572.717} C_VEL
LIN {X 0,Y 601.42,Z 449.57,A -85,B 0,C 180,E1 -575.117,E2 -575.117} C_VEL
LIN {X 0,Y 601.43,Z 449.564,A -85,B 0,C 180,E1 -577.42,E2 -577.42} C_VEL
LIN {X 0,Y 601.408,Z 449.563,A -85,B 0,C 180,E1 -579.996,E2 -579.996} C_VEL
LIN {X 0,Y 601.408,Z 449.57,A -85,B 0,C 180,E1 -582.671,E2 -582.671} C_VEL
LIN {X 0,Y 601.421,Z 449.565,A -85,B 0,C 180,E1 -585.483,E2 -585.483} C_VEL
LIN {X 0,Y 601.425,Z 449.564,A -85,B 0,C 180,E1 -588.407,E2 -588.407} C_VEL
LIN {X 0,Y 601.438,Z 449.569,A -85,B 0,C 180,E1 -590.877,E2 -590.877} C_VEL
LIN {X 0,Y 601.431,Z 449.561,A -85,B 0,C 180,E1 -593.736,E2 -593.736} C_VEL
LIN {X 0,Y 601.431,Z 449.56,A -85,B 0,C 180,E1 -596.065,E2 -596.065} C_VEL
LIN {X 0,Y 601.442,Z 449.563,A -85,B 0,C 180,E1 -598.543,E2 -598.543} C_VEL
LIN {X 0,Y 601.434,Z 449.566,A -85,B 0,C 180,E1 -601.374,E2 -601.374} C_VEL
LIN {X 0,Y 601.404,Z 449.567,A -85,B 0,C 180,E1 -603.637,E2 -603.637} C_VEL
LIN {X 0,Y 601.42,Z 449.565,A -85,B 0,C 180,E1 -606.59,E2 -606.59} C_VEL
LIN {X 0,Y 601.435,Z 449.567,A -85,B 0,C 180,E1 -609.479,E2 -609.479} C_VEL
LIN {X 0,Y 601.397,Z 449.564,A -85,B 0,C 180,E1 -612.312,E2 -612.312} C_VEL
LIN {X 0,Y 601.417,Z 449.564,A -85,B 0,C 180,E1 -614.409,E2 -614.409} C_VEL
LIN {X 0,Y 601.461,Z 449.765,A -85,B 0,C 180,E1 -617.066,E2 -617.066} C_VEL
LIN {X 0,Y 601.619,Z 450.57,A -85,B 0,C 180,E1 -617.155,E2 -617.155} C_VEL
LIN {X 0,Y 601.618,Z 534.984,A -85,B 0,C 180,E1 -618.204,E2 -618.204} C_VEL
LIN {X 0,Y 601.578,Z 548.666,A -85,B 0,C 180,E1 -618.524,E2 -618.524} C_VEL
LIN {X 0,Y 601.566,Z 560.226,A -85,B 0,C 180,E1 -618.921,E2 -618.921} C_VEL
LIN {X 0,Y 601.514,Z 572.384,A -85,B 0,C 180,E1 -619.481,E2 -619.481} C_VEL
LIN {X 0,Y 601.467,Z 583.805,A -85,B 0,C 180,E1 -620.161,E2 -620.161} C_VEL
LIN {X 0,Y 601.438,Z 594.095,A -85,B 0,C 180,E1 -620.924,E2 -620.924} C_VEL
LIN {X 0,Y 601.411,Z 603.357,A -85,B 0,C 180,E1 -621.77,E2 -621.77} C_VEL
LIN {X 0,Y 601.388,Z 612.329,A -85,B 0,C 180,E1 -622.783,E2 -622.783} C_VEL
LIN {X 0,Y 601.376,Z 619.468,A -85,B 0,C 180,E1 -623.781,E2 -623.781} C_VEL
LIN {X 0,Y 601.372,Z 624.438,A -85,B 0,C 180,E1 -624.636,E2 -624.636} C_VEL
LIN {X 0,Y 601.354,Z 629.181,A -85,B 0,C 180,E1 -625.643,E2 -625.643} C_VEL
LIN {X 0,Y 601.344,Z 632.815,A -85,B 0,C 180,E1 -626.65,E2 -626.65} C_VEL
LIN {X 0,Y 601.324,Z 634.693,A -85,B 0,C 180,E1 -627.321,E2 -627.321} C_VEL
LIN {X 0,Y 601.342,Z 636.127,A -85,B 0,C 180,E1 -627.991,E2 -627.991} C_VEL
LIN {X 0,Y 601.339,Z 637.753,A -85,B 0,C 180,E1 -629.33,E2 -629.33} C_VEL
LIN {X 0,Y 601.336,Z 637.996,A -85,B 0,C 180,E1 -630,E2 -630} C_VEL
LIN {X 0,Y 601.339,Z 637.815,A -85,B 0,C 180,E1 -630.67,E2 -630.67} C_VEL
LIN {X 0,Y 601.343,Z 636.276,A -85,B 0,C 180,E1 -632.009,E2 -632.009} C_VEL
LIN {X 0,Y 601.326,Z 634.917,A -85,B 0,C 180,E1 -632.679,E2 -632.679} C_VEL
LIN {X 0,Y 601.368,Z 632.04,A -85,B 0,C 180,E1 -633.685,E2 -633.685} C_VEL
LIN {X 0,Y 601.337,Z 628.141,A -85,B 0,C 180,E1 -634.693,E2 -634.693} C_VEL
LIN {X 0,Y 601.373,Z 623.11,A -85,B 0,C 180,E1 -635.701,E2 -635.701} C_VEL
LIN {X 0,Y 601.382,Z 616.792,A -85,B 0,C 180,E1 -636.711,E2 -636.711} C_VEL
LIN {X 0,Y 601.396,Z 608.875,A -85,B 0,C 180,E1 -637.723,E2 -637.723} C_VEL
LIN {X 0,Y 601.436,Z 599.032,A -85,B 0,C 180,E1 -638.737,E2 -638.737} C_VEL
LIN {X 0,Y 601.448,Z 588.712,A -85,B 0,C 180,E1 -639.585,E2 -639.585} C_VEL
LIN {X 0,Y 601.499,Z 577.093,A -85,B 0,C 180,E1 -640.349,E2 -640.349} C_VEL
LIN {X 0,Y 601.552,Z 565.849,A -85,B 0,C 180,E1 -640.93,E2 -640.93} C_VEL
LIN {X 0,Y 601.564,Z 553.438,A -85,B 0,C 180,E1 -641.416,E2 -641.416} C_VEL
LIN {X 0,Y 601.602,Z 540.551,A -85,B 0,C 180,E1 -641.775,E2 -641.775} C_VEL
LIN {X 0,Y 601.642,Z 528.273,A -85,B 0,C 180,E1 -641.988,E2 -641.988} C_VEL
LIN {X 0,Y 601.643,Z 450.654,A -85,B 0,C 180,E1 -642.93,E2 -642.93} C_VEL
LIN {X 0,Y 601.435,Z 449.637,A -85,B 0,C 180,E1 -643.064,E2 -643.064} C_VEL
LIN {X 0,Y 601.416,Z 449.565,A -85,B 0,C 180,E1 -645.591,E2 -645.591} C_VEL
LIN {X 0,Y 601.422,Z 449.563,A -85,B 0,C 180,E1 -648.391,E2 -648.391} C_VEL
LIN {X 0,Y 601.407,Z 449.57,A -85,B 0,C 180,E1 -651.239,E2 -651.239} C_VEL
LIN {X 0,Y 601.46,Z 449.558,A -85,B 0,C 180,E1 -654.14,E2 -654.14} C_VEL
LIN {X 0,Y 601.457,Z 449.566,A -85,B 0,C 180,E1 -657.11,E2 -657.11} C_VEL
LIN {X 0,Y 601.415,Z 449.568,A -85,B 0,C 180,E1 -659.393,E2 -659.393} C_VEL
LIN {X 0,Y 601.413,Z 449.564,A -85,B 0,C 180,E1 -661.725,E2 -661.725} C_VEL
LIN {X 0,Y 601.427,Z 449.562,A -85,B 0,C 180,E1 -664.117,E2 -664.117} C_VEL
LIN {X 0,Y 601.41,Z 449.567,A -85,B 0,C 180,E1 -666.581,E2 -666.581} C_VEL
LIN {X 0,Y 601.437,Z 449.564,A -85,B 0,C 180,E1 -669.535,E2 -669.535} C_VEL
LIN {X 0,Y 601.425,Z 449.563,A -85,B 0,C 180,E1 -671.764,E2 -671.764} C_VEL
LIN {X 0,Y 601.42,Z 449.565,A -85,B 0,C 180,E1 -674.534,E2 -674.534} C_VEL
LIN {X 0,Y 601.407,Z 449.57,A -85,B 0,C 180,E1 -677.408,E2 -677.408} C_VEL
LIN {X 0,Y 601.44,Z 449.56,A -85,B 0,C 180,E1 -680.463,E2 -680.463} C_VEL
LIN {X 0,Y 601.41,Z 449.571,A -85,B 0,C 180,E1 -683.417,E2 -683.417} C_VEL
LIN {X 0,Y 601.43,Z 449.562,A -85,B 0,C 180,E1 -686.063,E2 -686.063} C_VEL
LIN {X 0,Y 601.436,Z 449.561,A -85,B 0,C 180,E1 -688.541,E2 -688.541} C_VEL
LIN {X 0,Y 601.433,Z 449.569,A -85,B 0,C 180,E1 -691.373,E2 -691.373} C_VEL
LIN {X 0,Y 601.416,Z 449.564,A -85,B 0,C 180,E1 -694.129,E2 -694.129} C_VEL
LIN {X 0,Y 601.418,Z 449.564,A -85,B 0,C 180,E1 -696.589,E2 -696.589} C_VEL
LIN {X 0,Y 601.429,Z 449.569,A -85,B 0,C 180,E1 -699.478,E2 -699.478} C_VEL
LIN {X 0,Y 601.392,Z 449.566,A -85,B 0,C 180,E1 -702.311,E2 -702.311} C_VEL
LIN {X 0,Y 601.409,Z 449.564,A -85,B 0,C 180,E1 -704.408,E2 -704.408} C_VEL
LIN {X 0,Y 601.419,Z 449.571,A -85,B 0,C 180,E1 -707.172,E2 -707.172} C_VEL
LIN {X 0,Y 601.429,Z 449.564,A -85,B 0,C 180,E1 -709.905,E2 -709.905} C_VEL
LIN {X 0,Y 601.445,Z 449.56,A -85,B 0,C 180,E1 -712.615,E2 -712.615} C_VEL
LIN {X 0,Y 601.432,Z 449.571,A -85,B 0,C 180,E1 -715.308,E2 -715.308} C_VEL
LIN {X 0,Y 601.416,Z 449.565,A -85,B 0,C 180,E1 -717.991,E2 -717.991} C_VEL
LIN {X 0,Y 601.449,Z 449.56,A -85,B 0,C 180,E1 -720.669,E2 -720.669} C_VEL
LIN {X 0,Y 601.429,Z 449.57,A -85,B 0,C 180,E1 -723.35,E2 -723.35} C_VEL
LIN {X 0,Y 601.406,Z 449.567,A -85,B 0,C 180,E1 -726.037,E2 -726.037} C_VEL
LIN {X 0,Y 601.435,Z 449.562,A -85,B 0,C 180,E1 -728.738,E2 -728.738} C_VEL
LIN {X 0,Y 601.426,Z 449.572,A -85,B 0,C 180,E1 -731.458,E2 -731.458} C_VEL
LIN {X 0,Y 601.409,Z 449.566,A -85,B 0,C 180,E1 -734.206,E2 -734.206} C_VEL
LIN {X 0,Y 601.426,Z 449.564,A -85,B 0,C 180,E1 -736.986,E2 -736.986} C_VEL
LIN {X 0,Y 601.401,Z 449.572,A -85,B 0,C 180,E1 -739.81,E2 -739.81} C_VEL
LIN {X 0,Y 601.406,Z 449.565,A -85,B 0,C 180,E1 -742.606,E2 -742.606} C_VEL
LIN {X 0,Y 601.398,Z 449.566,A -85,B 0,C 180,E1 -744.879,E2 -744.879} C_VEL
LIN {X 0,Y 601.415,Z 449.57,A -85,B 0,C 180,E1 -747.868,E2 -747.868} C_VEL
LIN {X 0,Y 601.44,Z 449.563,A -85,B 0,C 180,E1 -750.163,E2 -750.163} C_VEL
LIN {X 0,Y 601.417,Z 449.563,A -85,B 0,C 180,E1 -752.717,E2 -752.717} C_VEL
LIN {X 0,Y 601.415,Z 449.565,A -85,B 0,C 180,E1 -755.116,E2 -755.116} C_VEL
LIN {X 0,Y 601.427,Z 449.568,A -85,B 0,C 180,E1 -757.42,E2 -757.42} C_VEL
LIN {X 0,Y 601.406,Z 449.571,A -85,B 0,C 180,E1 -759.996,E2 -759.996} C_VEL
LIN {X 0,Y 601.405,Z 449.564,A -85,B 0,C 180,E1 -762.671,E2 -762.671} C_VEL
LIN {X 0,Y 601.421,Z 449.568,A -85,B 0,C 180,E1 -765.483,E2 -765.483} C_VEL
LIN {X 0,Y 601.424,Z 449.564,A -85,B 0,C 180,E1 -768.407,E2 -768.407} C_VEL
LIN {X 0,Y 601.433,Z 449.561,A -85,B 0,C 180,E1 -770.876,E2 -770.876} C_VEL
LIN {X 0,Y 601.428,Z 449.571,A -85,B 0,C 180,E1 -773.736,E2 -773.736} C_VEL
LIN {X 0,Y 601.425,Z 449.563,A -85,B 0,C 180,E1 -776.687,E2 -776.687} C_VEL
LIN {X 0,Y 601.431,Z 449.562,A -85,B 0,C 180,E1 -779.059,E2 -779.059} C_VEL
LIN {X 0,Y 601.427,Z 449.565,A -85,B 0,C 180,E1 -781.374,E2 -781.374} C_VEL
LIN {X 0,Y 601.447,Z 449.741,A -85,B 0,C 180,E1 -783.616,E2 -783.616} C_VEL
LIN {X 0,Y 601.984,Z 452.995,A -85,B 0,C 180,E1 -784.021,E2 -784.021} C_VEL
LIN {X 0,Y 601.851,Z 478.518,A -85,B 0,C 180,E1 -786.808,E2 -786.808} C_VEL
LIN {X 0,Y 601.715,Z 505.246,A -85,B 0,C 180,E1 -789.667,E2 -789.667} C_VEL
LIN {X 0,Y 601.627,Z 530.46,A -85,B 0,C 180,E1 -792.319,E2 -792.319} C_VEL
LIN {X 0,Y 601.546,Z 557.356,A -85,B 0,C 180,E1 -795.106,E2 -795.106} C_VEL
LIN {X 0,Y 601.532,Z 574.142,A -85,B 0,C 180,E1 -796.799,E2 -796.799} C_VEL
LIN {X 0,Y 601.603,Z 683.962,A -85,B 0,C 180,E1 -798.14,E2 -798.14} C_VEL
LIN {X 0,Y 601.585,Z 697.227,A -85,B 0,C 180,E1 -798.438,E2 -798.438} C_VEL
LIN {X 0,Y 601.549,Z 708.927,A -85,B 0,C 180,E1 -798.826,E2 -798.826} C_VEL
LIN {X 0,Y 601.518,Z 719.928,A -85,B 0,C 180,E1 -799.311,E2 -799.311} C_VEL
LIN {X 0,Y 601.466,Z 730.584,A -85,B 0,C 180,E1 -799.906,E2 -799.906} C_VEL
LIN {X 0,Y 601.446,Z 741.478,A -85,B 0,C 180,E1 -800.67,E2 -800.67} C_VEL
LIN {X 0,Y 601.429,Z 752.114,A -85,B 0,C 180,E1 -801.601,E2 -801.601} C_VEL
LIN {X 0,Y 601.418,Z 759.962,A -85,B 0,C 180,E1 -802.446,E2 -802.446} C_VEL
LIN {X 0,Y 601.37,Z 767.225,A -85,B 0,C 180,E1 -803.398,E2 -803.398} C_VEL
LIN {X 0,Y 601.371,Z 772.867,A -85,B 0,C 180,E1 -804.299,E2 -804.299} C_VEL
LIN {X 0,Y 601.337,Z 777.951,A -85,B 0,C 180,E1 -805.307,E2 -805.307} C_VEL
LIN {X 0,Y 601.367,Z 781.896,A -85,B 0,C 180,E1 -806.315,E2 -806.315} C_VEL
LIN {X 0,Y 601.325,Z 784.809,A -85,B 0,C 180,E1 -807.321,E2 -807.321} C_VEL
LIN {X 0,Y 601.34,Z 786.202,A -85,B 0,C 180,E1 -807.991,E2 -807.991} C_VEL
LIN {X 0,Y 601.339,Z 787.784,A -85,B 0,C 180,E1 -809.33,E2 -809.33} C_VEL
LIN {X 0,Y 601.335,Z 788,A -85,B 0,C 180,E1 -810,E2 -810} C_VEL
LIN {X 0,Y 601.348,Z 787.184,A -85,B 0,C 180,E1 -811.339,E2 -811.339} C_VEL
LIN {X 0,Y 601.34,Z 786.202,A -85,B 0,C 180,E1 -812.009,E2 -812.009} C_VEL
LIN {X 0,Y 601.325,Z 784.809,A -85,B 0,C 180,E1 -812.679,E2 -812.679} C_VEL
LIN {X 0,Y 601.367,Z 781.896,A -85,B 0,C 180,E1 -813.685,E2 -813.685} C_VEL
LIN {X 0,Y 601.337,Z 777.95,A -85,B 0,C 180,E1 -814.693,E2 -814.693} C_VEL
LIN {X 0,Y 601.372,Z 771.878,A -85,B 0,C 180,E1 -815.869,E2 -815.869} C_VEL
LIN {X 0,Y 601.382,Z 765.237,A -85,B 0,C 180,E1 -816.88,E2 -816.88} C_VEL
LIN {X 0,Y 601.4,Z 756.991,A -85,B 0,C 180,E1 -817.892,E2 -817.892} C_VEL
LIN {X 0,Y 601.436,Z 748.539,A -85,B 0,C 180,E1 -818.737,E2 -818.737} C_VEL
LIN {X 0,Y 601.442,Z 738.095,A -85,B 0,C 180,E1 -819.585,E2 -819.585} C_VEL
LIN {X 0,Y 601.478,Z 727.761,A -85,B 0,C 180,E1 -820.264,E2 -820.264} C_VEL
LIN {X 0,Y 601.538,Z 716.899,A -85,B 0,C 180,E1 -820.836,E2 -820.836} C_VEL
LIN {X 0,Y 601.565,Z 704.38,A -85,B 0,C 180,E1 -821.34,E2 -821.34} C_VEL
LIN {X 0,Y 601.596,Z 691.364,A -85,B 0,C 180,E1 -821.711,E2 -821.711} C_VEL
LIN {X 0,Y 601.61,Z 678.106,A -85,B 0,C 180,E1 -821.946,E2 -821.946} C_VEL
LIN {X 0,Y 601.568,Z 574.557,A -85,B 0,C 180,E1 -823.19,E2 -823.19} C_VEL
LIN {X 0,Y 601.515,Z 573.349,A -85,B 0,C 180,E1 -823.255,E2 -823.255} C_VEL
LIN {X 0,Y 601.587,Z 545.589,A -85,B 0,C 180,E1 -826.108,E2 -826.108} C_VEL
LIN {X 0,Y 601.69,Z 517.012,A -85,B 0,C 180,E1 -829.089,E2 -829.089} C_VEL
LIN {X 0,Y 601.77,Z 490.117,A -85,B 0,C 180,E1 -831.945,E2 -831.945} C_VEL
LIN {X 0,Y 601.94,Z 464.596,A -85,B 0,C 180,E1 -834.704,E2 -834.704} C_VEL
LIN {X 0,Y 601.96,Z 452.014,A -85,B 0,C 180,E1 -836.088,E2 -836.088} C_VEL
LIN {X 0,Y 601.442,Z 449.659,A -85,B 0,C 180,E1 -836.408,E2 -836.408} C_VEL
LIN {X 0,Y 601.415,Z 449.565,A -85,B 0,C 180,E1 -839.393,E2 -839.393} C_VEL
LIN {X 0,Y 601.412,Z 449.568,A -85,B 0,C 180,E1 -841.725,E2 -841.725} C_VEL
LIN {X 0,Y 601.426,Z 449.573,A -85,B 0,C 180,E1 -844.118,E2 -844.118} C_VEL
LIN {X 0,Y 601.435,Z 449.561,A -85,B 0,C 180,E1 -847.382,E2 -847.382} C_VEL
LIN {X 0,Y 601.409,Z 449.572,A -85,B 0,C 180,E1 -849.994,E2 -849.994} C_VEL
LIN {X 0,Y 601.411,Z 449.568,A -85,B 0,C 180,E1 -852.669,E2 -852.669} C_VEL
LIN {X 0,Y 601.421,Z 449.563,A -85,B 0,C 180,E1 -855.481,E2 -855.481} C_VEL
LIN {X 0,Y 601.418,Z 449.572,A -85,B 0,C 180,E1 -858.406,E2 -858.406} C_VEL
LIN {X 0,Y 601.431,Z 449.563,A -85,B 0,C 180,E1 -860.875,E2 -860.875} C_VEL
LIN {X 0,Y 601.437,Z 449.563,A -85,B 0,C 180,E1 -863.733,E2 -863.733} C_VEL
LIN {X 0,Y 601.428,Z 449.568,A -85,B 0,C 180,E1 -866.063,E2 -866.063} C_VEL
LIN {X 0,Y 601.434,Z 449.569,A -85,B 0,C 180,E1 -868.541,E2 -868.541} C_VEL
LIN {X 0,Y 601.43,Z 449.561,A -85,B 0,C 180,E1 -871.373,E2 -871.373} C_VEL
LIN {X 0,Y 601.416,Z 449.569,A -85,B 0,C 180,E1 -874.129,E2 -874.129} C_VEL
LIN {X 0,Y 601.416,Z 449.571,A -85,B 0,C 180,E1 -876.589,E2 -876.589} C_VEL
LIN {X 0,Y 601.428,Z 449.561,A -85,B 0,C 180,E1 -879.478,E2 -879.478} C_VEL
LIN {X 0,Y 601.391,Z 449.574,A -85,B 0,C 180,E1 -882.311,E2 -882.311} C_VEL
LIN {X 0,Y 601.41,Z 449.574,A -85,B 0,C 180,E1 -884.409,E2 -884.409} C_VEL
LIN {X 0,Y 601.419,Z 449.564,A -85,B 0,C 180,E1 -887.172,E2 -887.172} C_VEL
LIN {X 0,Y 601.429,Z 449.563,A -85,B 0,C 180,E1 -889.905,E2 -889.905} C_VEL
LIN {X 0,Y 601.446,Z 449.569,A -85,B 0,C 180,E1 -892.615,E2 -892.615} C_VEL
LIN {X 0,Y 601.43,Z 449.562,A -85,B 0,C 180,E1 -895.308,E2 -895.308} C_VEL
LIN {X 0,Y 601.418,Z 449.565,A -85,B 0,C 180,E1 -897.991,E2 -897.991} C_VEL
LIN {X 0,Y 601.452,Z 449.569,A -85,B 0,C 180,E1 -900.67,E2 -900.67} C_VEL
LIN {X 0,Y 601.427,Z 449.563,A -85,B 0,C 180,E1 -903.35,E2 -903.35} C_VEL
LIN {X 0,Y 601.426,Z 449.564,A -85,B 0,C 180,E1 -906.037,E2 -906.037} C_VEL
LIN {X 0,Y 601.436,Z 449.57,A -85,B 0,C 180,E1 -908.738,E2 -908.738} C_VEL
LIN {X 0,Y 601.428,Z 449.562,A -85,B 0,C 180,E1 -911.458,E2 -911.458} C_VEL
LIN {X 0,Y 601.406,Z 449.568,A -85,B 0,C 180,E1 -912.39,E2 -912.39} C_VEL
LIN {X 0,Y 600.744,Z 449.656,A -85,B 0,C 180,E1 -912.95,E2 -912.95} C_VEL
LIN {X 0,Y 597.893,Z 450.011,A -85,B 0,C 180,E1 -913.858,E2 -913.858} C_VEL
LIN {X 0,Y 595.481,Z 450.311,A -85,B 0,C 180,E1 -914.588,E2 -914.588} C_VEL
LIN {X 0,Y 594.442,Z 450.435,A -85,B 0,C 180,E1 -915.151,E2 -915.151} C_VEL
LIN {X 0,Y 594.356,Z 450.444,A -85,B 0,C 180,E1 -915.342,E2 -915.342} C_VEL
LIN {X 0,Y 594.374,Z 450.441,A -85,B 0,C 180,E1 -917.904,E2 -917.904} C_VEL
LIN {X 0,Y 594.379,Z 450.448,A -85,B 0,C 180,E1 -920.92,E2 -920.92} C_VEL
LIN {X 0,Y 594.385,Z 450.439,A -85,B 0,C 180,E1 -923.704,E2 -923.704} C_VEL
LIN {X 0,Y 594.383,Z 450.449,A -85,B 0,C 180,E1 -926.7,E2 -926.7} C_VEL
LIN {X 0,Y 594.379,Z 450.446,A -85,B 0,C 180,E1 -928.999,E2 -928.999} C_VEL
LIN {X 0,Y 594.387,Z 450.438,A -85,B 0,C 180,E1 -931.646,E2 -931.646} C_VEL
LIN {X 0,Y 594.397,Z 450.443,A -85,B 0,C 180,E1 -934.579,E2 -934.579} C_VEL
LIN {X 0,Y 594.382,Z 450.447,A -85,B 0,C 180,E1 -937.087,E2 -937.087} C_VEL
LIN {X 0,Y 594.374,Z 450.439,A -85,B 0,C 180,E1 -939.776,E2 -939.776} C_VEL
LIN {X 0,Y 594.364,Z 450.444,A -85,B 0,C 180,E1 -942.376,E2 -942.376} C_VEL
LIN {X 0,Y 594.359,Z 450.449,A -85,B 0,C 180,E1 -945.192,E2 -945.192} C_VEL
LIN {X 0,Y 594.385,Z 450.44,A -85,B 0,C 180,E1 -947.627,E2 -947.627} C_VEL
LIN {X 0,Y 594.39,Z 450.44,A -85,B 0,C 180,E1 -950.322,E2 -950.322} C_VEL
LIN {X 0,Y 594.385,Z 450.448,A -85,B 0,C 180,E1 -952.914,E2 -952.914} C_VEL
LIN {X 0,Y 594.383,Z 450.437,A -85,B 0,C 180,E1 -955.862,E2 -955.862} C_VEL
LIN {X 0,Y 594.391,Z 450.442,A -85,B 0,C 180,E1 -958.652,E2 -958.652} C_VEL
LIN {X 0,Y 594.384,Z 450.45,A -85,B 0,C 180,E1 -961.043,E2 -961.043} C_VEL
LIN {X 0,Y 594.383,Z 450.439,A -85,B 0,C 180,E1 -963.979,E2 -963.979} C_VEL
LIN {X 0,Y 594.392,Z 450.439,A -85,B 0,C 180,E1 -966.297,E2 -966.297} C_VEL
LIN {X 0,Y 594.407,Z 450.447,A -85,B 0,C 180,E1 -969.225,E2 -969.225} C_VEL
LIN {X 0,Y 594.355,Z 450.44,A -85,B 0,C 180,E1 -972.095,E2 -972.095} C_VEL
LIN {X 0,Y 594.37,Z 450.442,A -85,B 0,C 180,E1 -974.22,E2 -974.22} C_VEL
LIN {X 0,Y 594.452,Z 450.592,A -85,B 0,C 180,E1 -976.911,E2 -976.911} C_VEL
LIN {X 0,Y 594.648,Z 451.704,A -85,B 0,C 180,E1 -977.024,E2 -977.024} C_VEL
LIN {X 0,Y 594.686,Z 533.871,A -85,B 0,C 180,E1 -978.043,E2 -978.043} C_VEL
LIN {X 0,Y 594.636,Z 547.168,A -85,B 0,C 180,E1 -978.345,E2 -978.345} C_VEL
LIN {X 0,Y 594.595,Z 559.16,A -85,B 0,C 180,E1 -978.748,E2 -978.748} C_VEL
LIN {X 0,Y 594.553,Z 570.769,A -85,B 0,C 180,E1 -979.271,E2 -979.271} C_VEL
LIN {X 0,Y 594.477,Z 582.535,A -85,B 0,C 180,E1 -979.958,E2 -979.958} C_VEL
LIN {X 0,Y 594.414,Z 593.044,A -85,B 0,C 180,E1 -980.73,E2 -980.73} C_VEL
LIN {X 0,Y 594.384,Z 601.649,A -85,B 0,C 180,E1 -981.501,E2 -981.501} C_VEL
LIN {X 0,Y 594.347,Z 609.575,A -85,B 0,C 180,E1 -982.356,E2 -982.356} C_VEL
LIN {X 0,Y 594.305,Z 617.395,A -85,B 0,C 180,E1 -983.39,E2 -983.39} C_VEL
LIN {X 0,Y 594.289,Z 624.442,A -85,B 0,C 180,E1 -984.571,E2 -984.571} C_VEL
LIN {X 0,Y 594.27,Z 629.184,A -85,B 0,C 180,E1 -985.591,E2 -985.591} C_VEL
LIN {X 0,Y 594.267,Z 632.817,A -85,B 0,C 180,E1 -986.61,E2 -986.61} C_VEL
LIN {X 0,Y 594.225,Z 634.695,A -85,B 0,C 180,E1 -987.288,E2 -987.288} C_VEL
LIN {X 0,Y 594.241,Z 636.127,A -85,B 0,C 180,E1 -987.967,E2 -987.967} C_VEL
LIN {X 0,Y 594.24,Z 637.753,A -85,B 0,C 180,E1 -989.322,E2 -989.322} C_VEL
LIN {X 0,Y 594.236,Z 637.996,A -85,B 0,C 180,E1 -990,E2 -990} C_VEL
LIN {X 0,Y 594.239,Z 637.815,A -85,B 0,C 180,E1 -990.678,E2 -990.678} C_VEL
LIN {X 0,Y 594.242,Z 636.276,A -85,B 0,C 180,E1 -992.033,E2 -992.033} C_VEL
LIN {X 0,Y 594.226,Z 634.915,A -85,B 0,C 180,E1 -992.712,E2 -992.712} C_VEL
LIN {X 0,Y 594.289,Z 632.038,A -85,B 0,C 180,E1 -993.729,E2 -993.729} C_VEL
LIN {X 0,Y 594.241,Z 628.139,A -85,B 0,C 180,E1 -994.749,E2 -994.749} C_VEL
LIN {X 0,Y 594.299,Z 623.108,A -85,B 0,C 180,E1 -995.769,E2 -995.769} C_VEL
LIN {X 0,Y 594.316,Z 616.789,A -85,B 0,C 180,E1 -996.791,E2 -996.791} C_VEL
LIN {X 0,Y 594.346,Z 608.87,A -85,B 0,C 180,E1 -997.815,E2 -997.815} C_VEL
LIN {X 0,Y 594.381,Z 599.025,A -85,B 0,C 180,E1 -998.842,E2 -998.842} C_VEL
LIN {X 0,Y 594.429,Z 588.707,A -85,B 0,C 180,E1 -999.699,E2 -999.699} C_VEL
LIN {X 0,Y 594.516,Z 577.081,A -85,B 0,C 180,E1 -1000.472,E2 -1000.472} C_VEL
LIN {X 0,Y 594.541,Z 565.257,A -85,B 0,C 180,E1 -1001.086,E2 -1001.086} C_VEL
LIN {X 0,Y 594.612,Z 552.242,A -85,B 0,C 180,E1 -1001.591,E2 -1001.591} C_VEL
LIN {X 0,Y 594.668,Z 539.611,A -85,B 0,C 180,E1 -1001.936,E2 -1001.936} C_VEL
LIN {X 0,Y 594.702,Z 526.476,A -85,B 0,C 180,E1 -1002.151,E2 -1002.151} C_VEL
LIN {X 0,Y 594.667,Z 451.79,A -85,B 0,C 180,E1 -1003.063,E2 -1003.063} C_VEL
LIN {X 0,Y 594.419,Z 450.61,A -85,B 0,C 180,E1 -1003.177,E2 -1003.177} C_VEL
LIN {X 0,Y 594.369,Z 450.443,A -85,B 0,C 180,E1 -1005.78,E2 -1005.78} C_VEL
LIN {X 0,Y 594.387,Z 450.441,A -85,B 0,C 180,E1 -1008.617,E2 -1008.617} C_VEL
LIN {X 0,Y 594.368,Z 450.443,A -85,B 0,C 180,E1 -1011.503,E2 -1011.503} C_VEL
LIN {X 0,Y 594.391,Z 450.442,A -85,B 0,C 180,E1 -1014.445,E2 -1014.445} C_VEL
LIN {X 0,Y 594.388,Z 450.445,A -85,B 0,C 180,E1 -1016.699,E2 -1016.699} C_VEL
LIN {X 0,Y 594.381,Z 450.45,A -85,B 0,C 180,E1 -1018.998,E2 -1018.998} C_VEL
LIN {X 0,Y 594.392,Z 450.44,A -85,B 0,C 180,E1 -1021.644,E2 -1021.644} C_VEL
LIN {X 0,Y 594.379,Z 450.444,A -85,B 0,C 180,E1 -1024.579,E2 -1024.579} C_VEL
LIN {X 0,Y 594.385,Z 450.449,A -85,B 0,C 180,E1 -1027.086,E2 -1027.086} C_VEL
LIN {X 0,Y 594.374,Z 450.442,A -85,B 0,C 180,E1 -1029.774,E2 -1029.774} C_VEL
LIN {X 0,Y 594.37,Z 450.441,A -85,B 0,C 180,E1 -1032.374,E2 -1032.374} C_VEL
LIN {X 0,Y 594.36,Z 450.452,A -85,B 0,C 180,E1 -1035.19,E2 -1035.19} C_VEL
LIN {X 0,Y 594.378,Z 450.44,A -85,B 0,C 180,E1 -1038.151,E2 -1038.151} C_VEL
LIN {X 0,Y 594.384,Z 450.449,A -85,B 0,C 180,E1 -1041.195,E2 -1041.195} C_VEL
LIN {X 0,Y 594.391,Z 450.441,A -85,B 0,C 180,E1 -1043.758,E2 -1043.758} C_VEL
LIN {X 0,Y 594.376,Z 450.44,A -85,B 0,C 180,E1 -1046.238,E2 -1046.238} C_VEL
LIN {X 0,Y 594.385,Z 450.44,A -85,B 0,C 180,E1 -1048.65,E2 -1048.65} C_VEL
LIN {X 0,Y 594.382,Z 450.445,A -85,B 0,C 180,E1 -1051.04,E2 -1051.04} C_VEL
LIN {X 0,Y 594.388,Z 450.44,A -85,B 0,C 180,E1 -1053.974,E2 -1053.974} C_VEL
LIN {X 0,Y 594.385,Z 450.439,A -85,B 0,C 180,E1 -1056.296,E2 -1056.296} C_VEL
LIN {X 0,Y 594.402,Z 450.447,A -85,B 0,C 180,E1 -1059.224,E2 -1059.224} C_VEL
LIN {X 0,Y 594.374,Z 450.441,A -85,B 0,C 180,E1 -1062.096,E2 -1062.096} C_VEL
LIN {X 0,Y 594.362,Z 450.442,A -85,B 0,C 180,E1 -1064.219,E2 -1064.219} C_VEL
LIN {X 0,Y 594.365,Z 450.447,A -85,B 0,C 180,E1 -1067.017,E2 -1067.017} C_VEL
LIN {X 0,Y 594.389,Z 450.442,A -85,B 0,C 180,E1 -1069.784,E2 -1069.784} C_VEL
LIN {X 0,Y 594.393,Z 450.438,A -85,B 0,C 180,E1 -1072.527,E2 -1072.527} C_VEL
LIN {X 0,Y 594.399,Z 450.446,A -85,B 0,C 180,E1 -1075.252,E2 -1075.252} C_VEL
LIN {X 0,Y 594.387,Z 450.441,A -85,B 0,C 180,E1 -1077.967,E2 -1077.967} C_VEL
LIN {X 0,Y 594.419,Z 450.435,A -85,B 0,C 180,E1 -1080.677,E2 -1080.677} C_VEL
LIN {X 0,Y 594.38,Z 450.449,A -85,B 0,C 180,E1 -1083.389,E2 -1083.389} C_VEL
LIN {X 0,Y 594.362,Z 450.444,A -85,B 0,C 180,E1 -1086.109,E2 -1086.109} C_VEL
LIN {X 0,Y 594.41,Z 450.437,A -85,B 0,C 180,E1 -1088.157,E2 -1088.157} C_VEL
LIN {X 0,Y 594.384,Z 450.442,A -85,B 0,C 180,E1 -1091.078,E2 -1091.078} C_VEL
LIN {X 0,Y 594.374,Z 450.449,A -85,B 0,C 180,E1 -1093.679,E2 -1093.679} C_VEL
LIN {X 0,Y 594.388,Z 450.439,A -85,B 0,C 180,E1 -1096.721,E2 -1096.721} C_VEL
LIN {X 0,Y 594.362,Z 450.447,A -85,B 0,C 180,E1 -1099.335,E2 -1099.335} C_VEL
LIN {X 0,Y 594.362,Z 450.451,A -85,B 0,C 180,E1 -1101.504,E2 -1101.504} C_VEL
LIN {X 0,Y 594.379,Z 450.44,A -85,B 0,C 180,E1 -1104.447,E2 -1104.447} C_VEL
LIN {X 0,Y 594.379,Z 450.439,A -85,B 0,C 180,E1 -1106.7,E2 -1106.7} C_VEL
LIN {X 0,Y 594.378,Z 450.441,A -85,B 0,C 180,E1 -1108.999,E2 -1108.999} C_VEL
LIN {X 0,Y 594.386,Z 450.45,A -85,B 0,C 180,E1 -1111.646,E2 -1111.646} C_VEL
LIN {X 0,Y 594.393,Z 450.438,A -85,B 0,C 180,E1 -1114.579,E2 -1114.579} C_VEL
LIN {X 0,Y 594.379,Z 450.442,A -85,B 0,C 180,E1 -1117.087,E2 -1117.087} C_VEL
LIN {X 0,Y 594.373,Z 450.452,A -85,B 0,C 180,E1 -1119.776,E2 -1119.776} C_VEL
LIN {X 0,Y 594.363,Z 450.443,A -85,B 0,C 180,E1 -1122.376,E2 -1122.376} C_VEL
LIN {X 0,Y 594.358,Z 450.443,A -85,B 0,C 180,E1 -1125.192,E2 -1125.192} C_VEL
LIN {X 0,Y 594.369,Z 450.449,A -85,B 0,C 180,E1 -1127.626,E2 -1127.626} C_VEL
LIN {X 0,Y 594.388,Z 450.442,A -85,B 0,C 180,E1 -1130.322,E2 -1130.322} C_VEL
LIN {X 0,Y 594.382,Z 450.44,A -85,B 0,C 180,E1 -1132.914,E2 -1132.914} C_VEL
LIN {X 0,Y 594.379,Z 450.451,A -85,B 0,C 180,E1 -1135.862,E2 -1135.862} C_VEL
LIN {X 0,Y 594.39,Z 450.439,A -85,B 0,C 180,E1 -1138.652,E2 -1138.652} C_VEL
LIN {X 0,Y 594.381,Z 450.441,A -85,B 0,C 180,E1 -1141.043,E2 -1141.043} C_VEL
LIN {X 0,Y 594.405,Z 450.668,A -85,B 0,C 180,E1 -1143.389,E2 -1143.389} C_VEL
LIN {X 0,Y 595.238,Z 455.351,A -85,B 0,C 180,E1 -1143.969,E2 -1143.969} C_VEL
LIN {X 0,Y 595.032,Z 480.031,A -85,B 0,C 180,E1 -1146.693,E2 -1146.693} C_VEL
LIN {X 0,Y 594.836,Z 506.927,A -85,B 0,C 180,E1 -1149.602,E2 -1149.602} C_VEL
LIN {X 0,Y 594.678,Z 533.822,A -85,B 0,C 180,E1 -1152.461,E2 -1152.461} C_VEL
LIN {X 0,Y 594.545,Z 560.718,A -85,B 0,C 180,E1 -1155.277,E2 -1155.277} C_VEL
LIN {X 0,Y 594.557,Z 574.136,A -85,B 0,C 180,E1 -1156.641,E2 -1156.641} C_VEL
LIN {X 0,Y 594.757,Z 585.112,A -85,B 0,C 180,E1 -1156.787,E2 -1156.787} C_VEL
LIN {X 0,Y 594.682,Z 683.962,A -85,B 0,C 180,E1 -1158,E2 -1158} C_VEL
LIN {X 0,Y 594.637,Z 696.468,A -85,B 0,C 180,E1 -1158.28,E2 -1158.28} C_VEL
LIN {X 0,Y 594.595,Z 709.575,A -85,B 0,C 180,E1 -1158.719,E2 -1158.719} C_VEL
LIN {X 0,Y 594.54,Z 721.638,A -85,B 0,C 180,E1 -1159.27,E2 -1159.27} C_VEL
LIN {X 0,Y 594.468,Z 733.203,A -85,B 0,C 180,E1 -1159.958,E2 -1159.958} C_VEL
LIN {X 0,Y 594.413,Z 743.599,A -85,B 0,C 180,E1 -1160.73,E2 -1160.73} C_VEL
LIN {X 0,Y 594.383,Z 752.114,A -85,B 0,C 180,E1 -1161.501,E2 -1161.501} C_VEL
LIN {X 0,Y 594.347,Z 759.962,A -85,B 0,C 180,E1 -1162.356,E2 -1162.356} C_VEL
LIN {X 0,Y 594.282,Z 767.813,A -85,B 0,C 180,E1 -1163.408,E2 -1163.408} C_VEL
LIN {X 0,Y 594.289,Z 774.681,A -85,B 0,C 180,E1 -1164.571,E2 -1164.571} C_VEL
LIN {X 0,Y 594.27,Z 779.372,A -85,B 0,C 180,E1 -1165.591,E2 -1165.591} C_VEL
LIN {X 0,Y 594.268,Z 782.956,A -85,B 0,C 180,E1 -1166.61,E2 -1166.61} C_VEL
LIN {X 0,Y 594.226,Z 784.809,A -85,B 0,C 180,E1 -1167.288,E2 -1167.288} C_VEL
LIN {X 0,Y 594.239,Z 786.202,A -85,B 0,C 180,E1 -1167.967,E2 -1167.967} C_VEL
LIN {X 0,Y 594.239,Z 787.784,A -85,B 0,C 180,E1 -1169.322,E2 -1169.322} C_VEL
LIN {X 0,Y 594.236,Z 788,A -85,B 0,C 180,E1 -1170,E2 -1170} C_VEL
LIN {X 0,Y 594.247,Z 787.185,A -85,B 0,C 180,E1 -1171.355,E2 -1171.355} C_VEL
LIN {X 0,Y 594.239,Z 786.202,A -85,B 0,C 180,E1 -1172.033,E2 -1172.033} C_VEL
LIN {X 0,Y 594.226,Z 784.81,A -85,B 0,C 180,E1 -1172.712,E2 -1172.712} C_VEL
LIN {X 0,Y 594.288,Z 781.896,A -85,B 0,C 180,E1 -1173.729,E2 -1173.729} C_VEL
LIN {X 0,Y 594.242,Z 777.95,A -85,B 0,C 180,E1 -1174.749,E2 -1174.749} C_VEL
LIN {X 0,Y 594.304,Z 771.878,A -85,B 0,C 180,E1 -1175.939,E2 -1175.939} C_VEL
LIN {X 0,Y 594.308,Z 765.237,A -85,B 0,C 180,E1 -1176.962,E2 -1176.962} C_VEL
LIN {X 0,Y 594.359,Z 756.991,A -85,B 0,C 180,E1 -1177.986,E2 -1177.986} C_VEL
LIN {X 0,Y 594.382,Z 748.539,A -85,B 0,C 180,E1 -1178.842,E2 -1178.842} C_VEL
LIN {X 0,Y 594.424,Z 738.096,A -85,B 0,C 180,E1 -1179.699,E2 -1179.699} C_VEL
LIN {X 0,Y 594.49,Z 727.763,A -85,B 0,C 180,E1 -1180.386,E2 -1180.386} C_VEL
LIN {X 0,Y 594.561,Z 716.688,A -85,B 0,C 180,E1 -1180.975,E2 -1180.975} C_VEL
LIN {X 0,Y 594.6,Z 704.707,A -85,B 0,C 180,E1 -1181.464,E2 -1181.464} C_VEL
LIN {X 0,Y 594.642,Z 691.363,A -85,B 0,C 180,E1 -1181.85,E2 -1181.85} C_VEL
LIN {X 0,Y 594.691,Z 678.106,A -85,B 0,C 180,E1 -1182.087,E2 -1182.087} C_VEL
LIN {X 0,Y 594.591,Z 574.545,A -85,B 0,C 180,E1 -1183.347,E2 -1183.347} C_VEL
LIN {X 0,Y 594.485,Z 573.349,A -85,B 0,C 180,E1 -1183.415,E2 -1183.415} C_VEL
LIN {X 0,Y 594.636,Z 545.589,A -85,B 0,C 180,E1 -1186.302,E2 -1186.302} C_VEL
LIN {X 0,Y 594.763,Z 518.99,A -85,B 0,C 180,E1 -1189.11,E2 -1189.11} C_VEL
LIN {X 0,Y 594.938,Z 491.798,A -85,B 0,C 180,E1 -1192.028,E2 -1192.028} C_VEL
LIN {X 0,Y 595.157,Z 466.431,A -85,B 0,C 180,E1 -1194.801,E2 -1194.801} C_VEL
LIN {X 0,Y 595.226,Z 453.964,A -85,B 0,C 180,E1 -1196.187,E2 -1196.187} C_VEL
LIN {X 0,Y 594.403,Z 450.56,A -85,B 0,C 180,E1 -1196.639,E2 -1196.639} C_VEL
LIN {X 0,Y 594.379,Z 450.441,A -85,B 0,C 180,E1 -1198.998,E2 -1198.998} C_VEL
LIN {X 0,Y 594.391,Z 450.442,A -85,B 0,C 180,E1 -1201.644,E2 -1201.644} C_VEL
LIN {X 0,Y 594.377,Z 450.444,A -85,B 0,C 180,E1 -1204.579,E2 -1204.579} C_VEL
LIN {X 0,Y 594.389,Z 450.441,A -85,B 0,C 180,E1 -1207.608,E2 -1207.608} C_VEL
LIN {X 0,Y 594.37,Z 450.445,A -85,B 0,C 180,E1 -1210.566,E2 -1210.566} C_VEL
LIN {X 0,Y 594.377,Z 450.441,A -85,B 0,C 180,E1 -1213.297,E2 -1213.297} C_VEL
LIN {X 0,Y 594.363,Z 450.451,A -85,B 0,C 180,E1 -1216.16,E2 -1216.16} C_VEL
LIN {X 0,Y 594.376,Z 450.447,A -85,B 0,C 180,E1 -1218.536,E2 -1218.536} C_VEL
LIN {X 0,Y 594.382,Z 450.439,A -85,B 0,C 180,E1 -1221.294,E2 -1221.294} C_VEL
LIN {X 0,Y 594.39,Z 450.441,A -85,B 0,C 180,E1 -1223.758,E2 -1223.758} C_VEL
LIN {X 0,Y 594.375,Z 450.45,A -85,B 0,C 180,E1 -1226.238,E2 -1226.238} C_VEL
LIN {X 0,Y 594.383,Z 450.445,A -85,B 0,C 180,E1 -1228.65,E2 -1228.65} C_VEL
LIN {X 0,Y 594.38,Z 450.441,A -85,B 0,C 180,E1 -1231.04,E2 -1231.04} C_VEL
LIN {X 0,Y 594.388,Z 450.442,A -85,B 0,C 180,E1 -1233.974,E2 -1233.974} C_VEL
LIN {X 0,Y 594.384,Z 450.448,A -85,B 0,C 180,E1 -1236.296,E2 -1236.296} C_VEL
LIN {X 0,Y 594.4,Z 450.437,A -85,B 0,C 180,E1 -1239.224,E2 -1239.224} C_VEL
LIN {X 0,Y 594.373,Z 450.444,A -85,B 0,C 180,E1 -1242.096,E2 -1242.096} C_VEL
LIN {X 0,Y 594.363,Z 450.448,A -85,B 0,C 180,E1 -1244.219,E2 -1244.219} C_VEL
LIN {X 0,Y 594.365,Z 450.444,A -85,B 0,C 180,E1 -1247.017,E2 -1247.017} C_VEL
LIN {X 0,Y 594.388,Z 450.439,A -85,B 0,C 180,E1 -1249.784,E2 -1249.784} C_VEL
LIN {X 0,Y 594.41,Z 450.447,A -85,B 0,C 180,E1 -1252.527,E2 -1252.527} C_VEL
LIN {X 0,Y 594.398,Z 450.438,A -85,B 0,C 180,E1 -1255.252,E2 -1255.252} C_VEL
LIN {X 0,Y 594.388,Z 450.44,A -85,B 0,C 180,E1 -1257.967,E2 -1257.967} C_VEL
LIN {X 0,Y 594.422,Z 450.444,A -85,B 0,C 180,E1 -1260.677,E2 -1260.677} C_VEL
LIN {X 0,Y 594.378,Z 450.44,A -85,B 0,C 180,E1 -1263.389,E2 -1263.389} C_VEL
LIN {X 0,Y 594.38,Z 450.442,A -85,B 0,C 180,E1 -1266.109,E2 -1266.109} C_VEL
LIN {X 0,Y 594.396,Z 450.445,A -85,B 0,C 180,E1 -1268.842,E2 -1268.842} C_VEL
LIN {X 0,Y 594.386,Z 450.439,A -85,B 0,C 180,E1 -1271.596,E2 -1271.596} C_VEL
LIN {X 0,Y 594.38,Z 450.445,A -85,B 0,C 180,E1 -1274.377,E2 -1274.377} C_VEL
LIN {X 0,Y 594.356,Z 450.444,A -85,B 0,C 180,E1 -1275.342,E2 -1275.342} C_VEL
LIN {X 0,Y 593.686,Z 450.528,A -85,B 0,C 180,E1 -1275.908,E2 -1275.908} C_VEL
LIN {X 0,Y 590.832,Z 450.891,A -85,B 0,C 180,E1 -1276.826,E2 -1276.826} C_VEL
LIN {X 0,Y 588.427,Z 451.186,A -85,B 0,C 180,E1 -1277.565,E2 -1277.565} C_VEL
LIN {X 0,Y 587.4,Z 451.311,A -85,B 0,C 180,E1 -1278.135,E2 -1278.135} C_VEL
LIN {X 0,Y 587.32,Z 451.322,A -85,B 0,C 180,E1 -1278.328,E2 -1278.328} C_VEL
LIN {X 0,Y 587.349,Z 451.321,A -85,B 0,C 180,E1 -1281.045,E2 -1281.045} C_VEL
LIN {X 0,Y 587.33,Z 451.318,A -85,B 0,C 180,E1 -1284.007,E2 -1284.007} C_VEL
LIN {X 0,Y 587.357,Z 451.317,A -85,B 0,C 180,E1 -1286.278,E2 -1286.278} C_VEL
LIN {X 0,Y 587.347,Z 451.319,A -85,B 0,C 180,E1 -1289.135,E2 -1289.135} C_VEL
LIN {X 0,Y 587.35,Z 451.313,A -85,B 0,C 180,E1 -1291.839,E2 -1291.839} C_VEL
LIN {X 0,Y 587.354,Z 451.317,A -85,B 0,C 180,E1 -1294.35,E2 -1294.35} C_VEL
LIN {X 0,Y 587.348,Z 451.324,A -85,B 0,C 180,E1 -1296.747,E2 -1296.747} C_VEL
LIN {X 0,Y 587.344,Z 451.317,A -85,B 0,C 180,E1 -1299.36,E2 -1299.36} C_VEL
LIN {X 0,Y 587.329,Z 451.318,A -85,B 0,C 180,E1 -1302.109,E2 -1302.109} C_VEL
LIN {X 0,Y 587.312,Z 451.328,A -85,B 0,C 180,E1 -1305.09,E2 -1305.09} C_VEL
LIN {X 0,Y 587.35,Z 451.314,A -85,B 0,C 180,E1 -1307.928,E2 -1307.928} C_VEL
LIN {X 0,Y 587.335,Z 451.327,A -85,B 0,C 180,E1 -1311.058,E2 -1311.058} C_VEL
LIN {X 0,Y 587.351,Z 451.319,A -85,B 0,C 180,E1 -1313.293,E2 -1313.293} C_VEL
LIN {X 0,Y 587.365,Z 451.31,A -85,B 0,C 180,E1 -1315.781,E2 -1315.781} C_VEL
LIN {X 0,Y 587.353,Z 451.315,A -85,B 0,C 180,E1 -1318.233,E2 -1318.233} C_VEL
LIN {X 0,Y 587.35,Z 451.323,A -85,B 0,C 180,E1 -1320.867,E2 -1320.867} C_VEL
LIN {X 0,Y 587.359,Z 451.315,A -85,B 0,C 180,E1 -1323.82,E2 -1323.82} C_VEL
LIN {X 0,Y 587.339,Z 451.318,A -85,B 0,C 180,E1 -1325.994,E2 -1325.994} C_VEL
LIN {X 0,Y 587.324,Z 451.318,A -85,B 0,C 180,E1 -1328.226,E2 -1328.226} C_VEL
LIN {X 0,Y 587.352,Z 451.323,A -85,B 0,C 180,E1 -1331.152,E2 -1331.152} C_VEL
LIN {X 0,Y 587.328,Z 451.32,A -85,B 0,C 180,E1 -1334.025,E2 -1334.025} C_VEL
LIN {X 0,Y 587.398,Z 451.521,A -85,B 0,C 180,E1 -1336.773,E2 -1336.773} C_VEL
LIN {X 0,Y 587.673,Z 452.677,A -85,B 0,C 180,E1 -1336.881,E2 -1336.881} C_VEL
LIN {X 0,Y 587.818,Z 483.316,A -85,B 0,C 180,E1 -1337.265,E2 -1337.265} C_VEL
LIN {X 0,Y 587.742,Z 533.901,A -85,B 0,C 180,E1 -1337.9,E2 -1337.9} C_VEL
LIN {X 0,Y 587.704,Z 547.189,A -85,B 0,C 180,E1 -1338.205,E2 -1338.205} C_VEL
LIN {X 0,Y 587.629,Z 559.751,A -85,B 0,C 180,E1 -1338.635,E2 -1338.635} C_VEL
LIN {X 0,Y 587.57,Z 570.783,A -85,B 0,C 180,E1 -1339.142,E2 -1339.142} C_VEL
LIN {X 0,Y 587.468,Z 582.541,A -85,B 0,C 180,E1 -1339.837,E2 -1339.837} C_VEL
LIN {X 0,Y 587.393,Z 593.053,A -85,B 0,C 180,E1 -1340.618,E2 -1340.618} C_VEL
LIN {X 0,Y 587.323,Z 601.655,A -85,B 0,C 180,E1 -1341.398,E2 -1341.398} C_VEL
LIN {X 0,Y 587.274,Z 609.579,A -85,B 0,C 180,E1 -1342.263,E2 -1342.263} C_VEL
LIN {X 0,Y 587.235,Z 616.149,A -85,B 0,C 180,E1 -1343.127,E2 -1343.127} C_VEL
LIN {X 0,Y 587.237,Z 622.619,A -85,B 0,C 180,E1 -1344.162,E2 -1344.162} C_VEL
LIN {X 0,Y 587.146,Z 627.759,A -85,B 0,C 180,E1 -1345.194,E2 -1345.194} C_VEL
LIN {X 0,Y 587.212,Z 631.748,A -85,B 0,C 180,E1 -1346.226,E2 -1346.226} C_VEL
LIN {X 0,Y 587.131,Z 634.698,A -85,B 0,C 180,E1 -1347.256,E2 -1347.256} C_VEL
LIN {X 0,Y 587.14,Z 636.127,A -85,B 0,C 180,E1 -1347.942,E2 -1347.942} C_VEL
LIN {X 0,Y 587.14,Z 637.754,A -85,B 0,C 180,E1 -1349.314,E2 -1349.314} C_VEL
LIN {X 0,Y 587.137,Z 637.996,A -85,B 0,C 180,E1 -1350,E2 -1350} C_VEL
LIN {X 0,Y 587.14,Z 637.815,A -85,B 0,C 180,E1 -1350.686,E2 -1350.686} C_VEL
LIN {X 0,Y 587.14,Z 636.274,A -85,B 0,C 180,E1 -1352.058,E2 -1352.058} C_VEL
LIN {X 0,Y 587.133,Z 634.914,A -85,B 0,C 180,E1 -1352.744,E2 -1352.744} C_VEL
LIN {X 0,Y 587.213,Z 632.036,A -85,B 0,C 180,E1 -1353.774,E2 -1353.774} C_VEL
LIN {X 0,Y 587.147,Z 628.136,A -85,B 0,C 180,E1 -1354.806,E2 -1354.806} C_VEL
LIN {X 0,Y 587.229,Z 623.105,A -85,B 0,C 180,E1 -1355.839,E2 -1355.839} C_VEL
LIN {X 0,Y 587.23,Z 616.785,A -85,B 0,C 180,E1 -1356.873,E2 -1356.873} C_VEL
LIN {X 0,Y 587.288,Z 608.865,A -85,B 0,C 180,E1 -1357.91,E2 -1357.91} C_VEL
LIN {X 0,Y 587.343,Z 599.018,A -85,B 0,C 180,E1 -1358.949,E2 -1358.949} C_VEL
LIN {X 0,Y 587.415,Z 588.702,A -85,B 0,C 180,E1 -1359.816,E2 -1359.816} C_VEL
LIN {X 0,Y 587.517,Z 578.498,A -85,B 0,C 180,E1 -1360.511,E2 -1360.511} C_VEL
LIN {X 0,Y 587.575,Z 566.282,A -85,B 0,C 180,E1 -1361.172,E2 -1361.172} C_VEL
LIN {X 0,Y 587.632,Z 553.596,A -85,B 0,C 180,E1 -1361.685,E2 -1361.685} C_VEL
LIN {X 0,Y 587.716,Z 540.504,A -85,B 0,C 180,E1 -1362.057,E2 -1362.057} C_VEL
LIN {X 0,Y 587.785,Z 528.194,A -85,B 0,C 180,E1 -1362.275,E2 -1362.275} C_VEL
LIN {X 0,Y 587.781,Z 453.198,A -85,B 0,C 180,E1 -1363.197,E2 -1363.197} C_VEL
LIN {X 0,Y 587.438,Z 451.819,A -85,B 0,C 180,E1 -1363.271,E2 -1363.271} C_VEL
LIN {X 0,Y 587.34,Z 451.345,A -85,B 0,C 180,E1 -1363.405,E2 -1363.405} C_VEL
LIN {X 0,Y 587.327,Z 451.32,A -85,B 0,C 180,E1 -1365.975,E2 -1365.975} C_VEL
LIN {X 0,Y 587.351,Z 451.321,A -85,B 0,C 180,E1 -1368.848,E2 -1368.848} C_VEL
LIN {X 0,Y 587.324,Z 451.318,A -85,B 0,C 180,E1 -1371.774,E2 -1371.774} C_VEL
LIN {X 0,Y 587.352,Z 451.323,A -85,B 0,C 180,E1 -1374.758,E2 -1374.758} C_VEL
LIN {X 0,Y 587.352,Z 451.314,A -85,B 0,C 180,E1 -1377.692,E2 -1377.692} C_VEL
LIN {X 0,Y 587.343,Z 451.32,A -85,B 0,C 180,E1 -1380.51,E2 -1380.51} C_VEL
LIN {X 0,Y 587.338,Z 451.327,A -85,B 0,C 180,E1 -1383.111,E2 -1383.111} C_VEL
LIN {X 0,Y 587.326,Z 451.321,A -85,B 0,C 180,E1 -1385.541,E2 -1385.541} C_VEL
LIN {X 0,Y 587.341,Z 451.317,A -85,B 0,C 180,E1 -1387.838,E2 -1387.838} C_VEL
LIN {X 0,Y 587.318,Z 451.32,A -85,B 0,C 180,E1 -1390.253,E2 -1390.253} C_VEL
LIN {X 0,Y 587.324,Z 451.328,A -85,B 0,C 180,E1 -1393.119,E2 -1393.119} C_VEL
LIN {X 0,Y 587.318,Z 451.32,A -85,B 0,C 180,E1 -1396.049,E2 -1396.049} C_VEL
LIN {X 0,Y 587.333,Z 451.324,A -85,B 0,C 180,E1 -1398.924,E2 -1398.924} C_VEL
LIN {X 0,Y 587.329,Z 451.322,A -85,B 0,C 180,E1 -1401.52,E2 -1401.52} C_VEL
LIN {X 0,Y 587.349,Z 451.317,A -85,B 0,C 180,E1 -1404.453,E2 -1404.453} C_VEL
LIN {X 0,Y 587.333,Z 451.323,A -85,B 0,C 180,E1 -1406.887,E2 -1406.887} C_VEL
LIN {X 0,Y 587.344,Z 451.319,A -85,B 0,C 180,E1 -1409.487,E2 -1409.487} C_VEL
LIN {X 0,Y 587.343,Z 451.316,A -85,B 0,C 180,E1 -1412.306,E2 -1412.306} C_VEL
LIN {X 0,Y 587.335,Z 451.318,A -85,B 0,C 180,E1 -1414.483,E2 -1414.483} C_VEL
LIN {X 0,Y 587.333,Z 451.324,A -85,B 0,C 180,E1 -1417.486,E2 -1417.486} C_VEL
LIN {X 0,Y 587.327,Z 451.323,A -85,B 0,C 180,E1 -1419.695,E2 -1419.695} C_VEL
LIN {X 0,Y 587.351,Z 451.316,A -85,B 0,C 180,E1 -1422.594,E2 -1422.594} C_VEL
LIN {X 0,Y 587.354,Z 451.319,A -85,B 0,C 180,E1 -1425.739,E2 -1425.739} C_VEL
LIN {X 0,Y 587.352,Z 451.318,A -85,B 0,C 180,E1 -1428.858,E2 -1428.858} C_VEL
LIN {X 0,Y 587.364,Z 451.318,A -85,B 0,C 180,E1 -1431.745,E2 -1431.745} C_VEL
LIN {X 0,Y 587.352,Z 451.315,A -85,B 0,C 180,E1 -1434.507,E2 -1434.507} C_VEL
LIN {X 0,Y 587.376,Z 451.319,A -85,B 0,C 180,E1 -1437.257,E2 -1437.257} C_VEL
LIN {X 0,Y 587.373,Z 451.315,A -85,B 0,C 180,E1 -1440,E2 -1440} C_VEL
LIN {X 0,Y 587.375,Z 451.313,A -85,B 0,C 180,E1 -1442.743,E2 -1442.743} C_VEL
LIN {X 0,Y 587.352,Z 451.325,A -85,B 0,C 180,E1 -1445.493,E2 -1445.493} C_VEL
LIN {X 0,Y 587.363,Z 451.315,A -85,B 0,C 180,E1 -1448.255,E2 -1448.255} C_VEL
LIN {X 0,Y 587.352,Z 451.319,A -85,B 0,C 180,E1 -1451.142,E2 -1451.142} C_VEL
LIN {X 0,Y 587.354,Z 451.316,A -85,B 0,C 180,E1 -1454.261,E2 -1454.261} C_VEL
LIN {X 0,Y 587.35,Z 451.323,A -85,B 0,C 180,E1 -1457.406,E2 -1457.406} C_VEL
LIN {X 0,Y 587.325,Z 451.319,A -85,B 0,C 180,E1 -1460.305,E2 -1460.305} C_VEL
LIN {X 0,Y 587.315,Z 451.325,A -85,B 0,C 180,E1 -1463.259,E2 -1463.259} C_VEL
LIN {X 0,Y 587.333,Z 451.326,A -85,B 0,C 180,E1 -1465.517,E2 -1465.517} C_VEL
LIN {X 0,Y 587.341,Z 451.324,A -85,B 0,C 180,E1 -1467.818,E2 -1467.818} C_VEL
LIN {X 0,Y 587.343,Z 451.317,A -85,B 0,C 180,E1 -1470.513,E2 -1470.513} C_VEL
LIN {X 0,Y 587.33,Z 451.323,A -85,B 0,C 180,E1 -1473.397,E2 -1473.397} C_VEL
LIN {X 0,Y 587.351,Z 451.323,A -85,B 0,C 180,E1 -1475.896,E2 -1475.896} C_VEL
LIN {X 0,Y 587.327,Z 451.319,A -85,B 0,C 180,E1 -1478.48,E2 -1478.48} C_VEL
LIN {X 0,Y 587.331,Z 451.32,A -85,B 0,C 180,E1 -1481.158,E2 -1481.158} C_VEL
LIN {X 0,Y 587.321,Z 451.323,A -85,B 0,C 180,E1 -1484.114,E2 -1484.114} C_VEL
LIN {X 0,Y 587.319,Z 451.32,A -85,B 0,C 180,E1 -1486.995,E2 -1486.995} C_VEL
LIN {X 0,Y 587.317,Z 451.328,A -85,B 0,C 180,E1 -1489.747,E2 -1489.747} C_VEL
LIN {X 0,Y 587.344,Z 451.319,A -85,B 0,C 180,E1 -1492.393,E2 -1492.393} C_VEL
LIN {X 0,Y 587.346,Z 451.324,A -85,B 0,C 180,E1 -1495.653,E2 -1495.653} C_VEL
LIN {X 0,Y 587.351,Z 451.32,A -85,B 0,C 180,E1 -1498.233,E2 -1498.233} C_VEL
LIN {X 0,Y 587.348,Z 451.318,A -85,B 0,C 180,E1 -1500.867,E2 -1500.867} C_VEL
LIN {X 0,Y 587.357,Z 451.514,A -85,B 0,C 180,E1 -1503.136,E2 -1503.136} C_VEL
LIN {X 0,Y 588.459,Z 456.498,A -85,B 0,C 180,E1 -1503.776,E2 -1503.776} C_VEL
LIN {X 0,Y 588.248,Z 480.031,A -85,B 0,C 180,E1 -1506.408,E2 -1506.408} C_VEL
LIN {X 0,Y 587.976,Z 506.927,A -85,B 0,C 180,E1 -1509.354,E2 -1509.354} C_VEL
LIN {X 0,Y 587.751,Z 533.822,A -85,B 0,C 180,E1 -1512.247,E2 -1512.247} C_VEL
LIN {X 0,Y 587.592,Z 560.718,A -85,B 0,C 180,E1 -1515.099,E2 -1515.099} C_VEL
LIN {X 0,Y 587.53,Z 574.13,A -85,B 0,C 180,E1 -1516.478,E2 -1516.478} C_VEL
LIN {X 0,Y 587.871,Z 579.746,A -85,B 0,C 180,E1 -1516.563,E2 -1516.563} C_VEL
LIN {X 0,Y 587.745,Z 683.962,A -85,B 0,C 180,E1 -1517.856,E2 -1517.856} C_VEL
LIN {X 0,Y 587.682,Z 696.468,A -85,B 0,C 180,E1 -1518.139,E2 -1518.139} C_VEL
LIN {X 0,Y 587.627,Z 709.757,A -85,B 0,C 180,E1 -1518.59,E2 -1518.59} C_VEL
LIN {X 0,Y 587.555,Z 721.636,A -85,B 0,C 180,E1 -1519.141,E2 -1519.141} C_VEL
LIN {X 0,Y 587.465,Z 733.204,A -85,B 0,C 180,E1 -1519.837,E2 -1519.837} C_VEL
LIN {X 0,Y 587.391,Z 743.6,A -85,B 0,C 180,E1 -1520.618,E2 -1520.618} C_VEL
LIN {X 0,Y 587.321,Z 752.114,A -85,B 0,C 180,E1 -1521.398,E2 -1521.398} C_VEL
LIN {X 0,Y 587.273,Z 759.962,A -85,B 0,C 180,E1 -1522.263,E2 -1522.263} C_VEL
LIN {X 0,Y 587.23,Z 766.471,A -85,B 0,C 180,E1 -1523.127,E2 -1523.127} C_VEL
LIN {X 0,Y 587.236,Z 772.867,A -85,B 0,C 180,E1 -1524.161,E2 -1524.161} C_VEL
LIN {X 0,Y 587.147,Z 777.95,A -85,B 0,C 180,E1 -1525.194,E2 -1525.194} C_VEL
LIN {X 0,Y 587.212,Z 781.896,A -85,B 0,C 180,E1 -1526.226,E2 -1526.226} C_VEL
LIN {X 0,Y 587.132,Z 784.809,A -85,B 0,C 180,E1 -1527.256,E2 -1527.256} C_VEL
LIN {X 0,Y 587.138,Z 786.201,A -85,B 0,C 180,E1 -1527.942,E2 -1527.942} C_VEL
LIN {X 0,Y 587.14,Z 787.784,A -85,B 0,C 180,E1 -1529.314,E2 -1529.314} C_VEL
LIN {X 0,Y 587.137,Z 788,A -85,B 0,C 180,E1 -1530,E2 -1530} C_VEL
LIN {X 0,Y 587.147,Z 787.185,A -85,B 0,C 180,E1 -1531.372,E2 -1531.372} C_VEL
LIN {X 0,Y 587.138,Z 786.201,A -85,B 0,C 180,E1 -1532.058,E2 -1532.058} C_VEL
LIN {X 0,Y 587.132,Z 784.81,A -85,B 0,C 180,E1 -1532.744,E2 -1532.744} C_VEL
LIN {X 0,Y 587.212,Z 781.896,A -85,B 0,C 180,E1 -1533.774,E2 -1533.774} C_VEL
LIN {X 0,Y 587.147,Z 777.95,A -85,B 0,C 180,E1 -1534.806,E2 -1534.806} C_VEL
LIN {X 0,Y 587.217,Z 771.878,A -85,B 0,C 180,E1 -1536.011,E2 -1536.011} C_VEL
LIN {X 0,Y 587.245,Z 765.238,A -85,B 0,C 180,E1 -1537.046,E2 -1537.046} C_VEL
LIN {X 0,Y 587.299,Z 756.992,A -85,B 0,C 180,E1 -1538.083,E2 -1538.083} C_VEL
LIN {X 0,Y 587.343,Z 748.54,A -85,B 0,C 180,E1 -1538.949,E2 -1538.949} C_VEL
LIN {X 0,Y 587.411,Z 738.098,A -85,B 0,C 180,E1 -1539.816,E2 -1539.816} C_VEL
LIN {X 0,Y 587.492,Z 727.763,A -85,B 0,C 180,E1 -1540.511,E2 -1540.511} C_VEL
LIN {X 0,Y 587.584,Z 715.804,A -85,B 0,C 180,E1 -1541.149,E2 -1541.149} C_VEL
LIN {X 0,Y 587.634,Z 703.597,A -85,B 0,C 180,E1 -1541.639,E2 -1541.639} C_VEL
LIN {X 0,Y 587.681,Z 690.448,A -85,B 0,C 180,E1 -1542.014,E2 -1542.014} C_VEL
LIN {X 0,Y 587.758,Z 678.106,A -85,B 0,C 180,E1 -1542.232,E2 -1542.232} C_VEL
LIN {X 0,Y 587.814,Z 576.169,A -85,B 0,C 180,E1 -1543.482,E2 -1543.482} C_VEL
LIN {X 0,Y 587.494,Z 573.578,A -85,B 0,C 180,E1 -1543.556,E2 -1543.556} C_VEL
LIN {X 0,Y 587.683,Z 547.27,A -85,B 0,C 180,E1 -1546.321,E2 -1546.321} C_VEL
LIN {X 0,Y 587.85,Z 520.488,A -85,B 0,C 180,E1 -1549.182,E2 -1549.182} C_VEL
LIN {X 0,Y 588.058,Z 495.16,A -85,B 0,C 180,E1 -1551.93,E2 -1551.93} C_VEL
LIN {X 0,Y 588.316,Z 471.626,A -85,B 0,C 180,E1 -1554.526,E2 -1554.526} C_VEL
LIN {X 0,Y 588.47,Z 456.498,A -85,B 0,C 180,E1 -1556.224,E2 -1556.224} C_VEL
LIN {X 0,Y 587.349,Z 451.466,A -85,B 0,C 180,E1 -1556.876,E2 -1556.876} C_VEL
LIN {X 0,Y 587.345,Z 451.319,A -85,B 0,C 180,E1 -1559.379,E2 -1559.379} C_VEL
LIN {X 0,Y 587.354,Z 451.321,A -85,B 0,C 180,E1 -1561.837,E2 -1561.837} C_VEL
LIN {X 0,Y 587.345,Z 451.324,A -85,B 0,C 180,E1 -1564.347,E2 -1564.347} C_VEL
LIN {X 0,Y 587.345,Z 451.318,A -85,B 0,C 180,E1 -1567.607,E2 -1567.607} C_VEL
LIN {X 0,Y 587.317,Z 451.329,A -85,B 0,C 180,E1 -1570.253,E2 -1570.253} C_VEL
LIN {X 0,Y 587.323,Z 451.32,A -85,B 0,C 180,E1 -1573.119,E2 -1573.119} C_VEL
LIN {X 0,Y 587.318,Z 451.326,A -85,B 0,C 180,E1 -1576.049,E2 -1576.049} C_VEL
LIN {X 0,Y 587.331,Z 451.32,A -85,B 0,C 180,E1 -1578.924,E2 -1578.924} C_VEL
LIN {X 0,Y 587.327,Z 451.319,A -85,B 0,C 180,E1 -1581.52,E2 -1581.52} C_VEL
LIN {X 0,Y 587.347,Z 451.324,A -85,B 0,C 180,E1 -1584.454,E2 -1584.454} C_VEL
LIN {X 0,Y 587.333,Z 451.319,A -85,B 0,C 180,E1 -1586.887,E2 -1586.887} C_VEL
LIN {X 0,Y 587.343,Z 451.317,A -85,B 0,C 180,E1 -1589.487,E2 -1589.487} C_VEL
LIN {X 0,Y 587.343,Z 451.326,A -85,B 0,C 180,E1 -1592.306,E2 -1592.306} C_VEL
LIN {X 0,Y 587.334,Z 451.327,A -85,B 0,C 180,E1 -1594.483,E2 -1594.483} C_VEL
LIN {X 0,Y 587.332,Z 451.318,A -85,B 0,C 180,E1 -1597.486,E2 -1597.486} C_VEL
LIN {X 0,Y 587.325,Z 451.318,A -85,B 0,C 180,E1 -1599.695,E2 -1599.695} C_VEL
LIN {X 0,Y 587.35,Z 451.323,A -85,B 0,C 180,E1 -1602.594,E2 -1602.594} C_VEL
LIN {X 0,Y 587.354,Z 451.316,A -85,B 0,C 180,E1 -1605.739,E2 -1605.739} C_VEL
LIN {X 0,Y 587.352,Z 451.319,A -85,B 0,C 180,E1 -1608.858,E2 -1608.858} C_VEL
LIN {X 0,Y 587.363,Z 451.315,A -85,B 0,C 180,E1 -1611.745,E2 -1611.745} C_VEL
LIN {X 0,Y 587.354,Z 451.325,A -85,B 0,C 180,E1 -1614.507,E2 -1614.507} C_VEL
LIN {X 0,Y 587.375,Z 451.313,A -85,B 0,C 180,E1 -1617.257,E2 -1617.257} C_VEL
LIN {X 0,Y 587.373,Z 451.315,A -85,B 0,C 180,E1 -1620,E2 -1620} C_VEL
LIN {X 0,Y 587.376,Z 451.32,A -85,B 0,C 180,E1 -1622.743,E2 -1622.743} C_VEL
LIN {X 0,Y 587.355,Z 451.315,A -85,B 0,C 180,E1 -1625.493,E2 -1625.493} C_VEL
LIN {X 0,Y 587.364,Z 451.318,A -85,B 0,C 180,E1 -1628.255,E2 -1628.255} C_VEL
LIN {X 0,Y 587.352,Z 451.319,A -85,B 0,C 180,E1 -1631.142,E2 -1631.142} C_VEL
LIN {X 0,Y 587.354,Z 451.319,A -85,B 0,C 180,E1 -1634.261,E2 -1634.261} C_VEL
LIN {X 0,Y 587.351,Z 451.316,A -85,B 0,C 180,E1 -1637.406,E2 -1637.406} C_VEL
LIN {X 0,Y 587.32,Z 451.322,A -85,B 0,C 180,E1 -1638.328,E2 -1638.328} C_VEL
LIN {X 0,Y 586.668,Z 451.409,A -85,B 0,C 180,E1 -1638.9,E2 -1638.9} C_VEL
LIN {X 0,Y 583.837,Z 451.762,A -85,B 0,C 180,E1 -1639.828,E2 -1639.828} C_VEL
LIN {X 0,Y 581.426,Z 452.061,A -85,B 0,C 180,E1 -1640.575,E2 -1640.575} C_VEL
LIN {X 0,Y 580.373,Z 452.189,A -85,B 0,C 180,E1 -1641.152,E2 -1641.152} C_VEL
LIN {X 0,Y 580.278,Z 452.198,A -85,B 0,C 180,E1 -1641.347,E2 -1641.347} C_VEL
LIN {X 0,Y 580.293,Z 452.198,A -85,B 0,C 180,E1 -1644.317,E2 -1644.317} C_VEL
LIN {X 0,Y 580.301,Z 452.201,A -85,B 0,C 180,E1 -1646.622,E2 -1646.622} C_VEL
LIN {X 0,Y 580.301,Z 452.193,A -85,B 0,C 180,E1 -1649.312,E2 -1649.312} C_VEL
LIN {X 0,Y 580.297,Z 452.192,A -85,B 0,C 180,E1 -1652.201,E2 -1652.201} C_VEL
LIN {X 0,Y 580.298,Z 452.201,A -85,B 0,C 180,E1 -1654.696,E2 -1654.696} C_VEL
LIN {X 0,Y 580.295,Z 452.198,A -85,B 0,C 180,E1 -1657.269,E2 -1657.269} C_VEL
LIN {X 0,Y 580.294,Z 452.192,A -85,B 0,C 180,E1 -1660.272,E2 -1660.272} C_VEL
LIN {X 0,Y 580.277,Z 452.202,A -85,B 0,C 180,E1 -1662.707,E2 -1662.707} C_VEL
LIN {X 0,Y 580.27,Z 452.198,A -85,B 0,C 180,E1 -1665.609,E2 -1665.609} C_VEL
LIN {X 0,Y 580.311,Z 452.191,A -85,B 0,C 180,E1 -1668.235,E2 -1668.235} C_VEL
LIN {X 0,Y 580.29,Z 452.206,A -85,B 0,C 180,E1 -1670.967,E2 -1670.967} C_VEL
LIN {X 0,Y 580.278,Z 452.195,A -85,B 0,C 180,E1 -1673.598,E2 -1673.598} C_VEL
LIN {X 0,Y 580.317,Z 452.187,A -85,B 0,C 180,E1 -1676.146,E2 -1676.146} C_VEL
LIN {X 0,Y 580.289,Z 452.198,A -85,B 0,C 180,E1 -1678.616,E2 -1678.616} C_VEL
LIN {X 0,Y 580.293,Z 452.205,A -85,B 0,C 180,E1 -1681.025,E2 -1681.025} C_VEL
LIN {X 0,Y 580.292,Z 452.196,A -85,B 0,C 180,E1 -1683.667,E2 -1683.667} C_VEL
LIN {X 0,Y 580.303,Z 452.196,A -85,B 0,C 180,E1 -1685.684,E2 -1685.684} C_VEL
LIN {X 0,Y 580.275,Z 452.196,A -85,B 0,C 180,E1 -1687.948,E2 -1687.948} C_VEL
LIN {X 0,Y 580.322,Z 452.198,A -85,B 0,C 180,E1 -1690.915,E2 -1690.915} C_VEL
LIN {X 0,Y 580.282,Z 452.2,A -85,B 0,C 180,E1 -1693.826,E2 -1693.826} C_VEL
LIN {X 0,Y 580.337,Z 452.357,A -85,B 0,C 180,E1 -1696.609,E2 -1696.609} C_VEL
LIN {X 0,Y 580.523,Z 453.241,A -85,B 0,C 180,E1 -1696.713,E2 -1696.713} C_VEL
LIN {X 0,Y 580.961,Z 454.748,A -85,B 0,C 180,E1 -1696.757,E2 -1696.757} C_VEL
LIN {X 0,Y 580.824,Z 533.931,A -85,B 0,C 180,E1 -1697.753,E2 -1697.753} C_VEL
LIN {X 0,Y 580.757,Z 547.208,A -85,B 0,C 180,E1 -1698.062,E2 -1698.062} C_VEL
LIN {X 0,Y 580.677,Z 559.367,A -85,B 0,C 180,E1 -1698.481,E2 -1698.481} C_VEL
LIN {X 0,Y 580.593,Z 570.796,A -85,B 0,C 180,E1 -1699.009,E2 -1699.009} C_VEL
LIN {X 0,Y 580.451,Z 582.546,A -85,B 0,C 180,E1 -1699.713,E2 -1699.713} C_VEL
LIN {X 0,Y 580.345,Z 593.062,A -85,B 0,C 180,E1 -1700.503,E2 -1700.503} C_VEL
LIN {X 0,Y 580.272,Z 601.661,A -85,B 0,C 180,E1 -1701.292,E2 -1701.292} C_VEL
LIN {X 0,Y 580.222,Z 609.584,A -85,B 0,C 180,E1 -1702.168,E2 -1702.168} C_VEL
LIN {X 0,Y 580.168,Z 617.285,A -85,B 0,C 180,E1 -1703.21,E2 -1703.21} C_VEL
LIN {X 0,Y 580.165,Z 622.622,A -85,B 0,C 180,E1 -1704.09,E2 -1704.09} C_VEL
LIN {X 0,Y 580.053,Z 627.761,A -85,B 0,C 180,E1 -1705.135,E2 -1705.135} C_VEL
LIN {X 0,Y 580.109,Z 631.75,A -85,B 0,C 180,E1 -1706.18,E2 -1706.18} C_VEL
LIN {X 0,Y 580.043,Z 634.7,A -85,B 0,C 180,E1 -1707.222,E2 -1707.222} C_VEL
LIN {X 0,Y 580.039,Z 636.127,A -85,B 0,C 180,E1 -1707.917,E2 -1707.917} C_VEL
LIN {X 0,Y 580.041,Z 637.755,A -85,B 0,C 180,E1 -1709.306,E2 -1709.306} C_VEL
LIN {X 0,Y 580.038,Z 637.996,A -85,B 0,C 180,E1 -1710,E2 -1710} C_VEL
LIN {X 0,Y 580.04,Z 637.815,A -85,B 0,C 180,E1 -1710.694,E2 -1710.694} C_VEL
LIN {X 0,Y 580.04,Z 636.273,A -85,B 0,C 180,E1 -1712.083,E2 -1712.083} C_VEL
LIN {X 0,Y 580.044,Z 634.912,A -85,B 0,C 180,E1 -1712.778,E2 -1712.778} C_VEL
LIN {X 0,Y 580.11,Z 632.034,A -85,B 0,C 180,E1 -1713.82,E2 -1713.82} C_VEL
LIN {X 0,Y 580.053,Z 628.134,A -85,B 0,C 180,E1 -1714.865,E2 -1714.865} C_VEL
LIN {X 0,Y 580.162,Z 623.103,A -85,B 0,C 180,E1 -1715.91,E2 -1715.91} C_VEL
LIN {X 0,Y 580.157,Z 616.781,A -85,B 0,C 180,E1 -1716.958,E2 -1716.958} C_VEL
LIN {X 0,Y 580.242,Z 608.86,A -85,B 0,C 180,E1 -1718.007,E2 -1718.007} C_VEL
LIN {X 0,Y 580.308,Z 599.012,A -85,B 0,C 180,E1 -1719.058,E2 -1719.058} C_VEL
LIN {X 0,Y 580.419,Z 588.697,A -85,B 0,C 180,E1 -1719.936,E2 -1719.936} C_VEL
LIN {X 0,Y 580.543,Z 577.058,A -85,B 0,C 180,E1 -1720.727,E2 -1720.727} C_VEL
LIN {X 0,Y 580.612,Z 565.508,A -85,B 0,C 180,E1 -1721.343,E2 -1721.343} C_VEL
LIN {X 0,Y 580.705,Z 553.51,A -85,B 0,C 180,E1 -1721.828,E2 -1721.828} C_VEL
LIN {X 0,Y 580.785,Z 540.481,A -85,B 0,C 180,E1 -1722.203,E2 -1722.203} C_VEL
LIN {X 0,Y 580.855,Z 528.154,A -85,B 0,C 180,E1 -1722.424,E2 -1722.424} C_VEL
LIN {X 0,Y 580.799,Z 454.218,A -85,B 0,C 180,E1 -1723.344,E2 -1723.344} C_VEL
LIN {X 0,Y 580.414,Z 452.798,A -85,B 0,C 180,E1 -1723.412,E2 -1723.412} C_VEL
LIN {X 0,Y 580.313,Z 452.216,A -85,B 0,C 180,E1 -1723.57,E2 -1723.57} C_VEL
LIN {X 0,Y 580.28,Z 452.199,A -85,B 0,C 180,E1 -1726.174,E2 -1726.174} C_VEL
LIN {X 0,Y 580.325,Z 452.198,A -85,B 0,C 180,E1 -1729.157,E2 -1729.157} C_VEL
LIN {X 0,Y 580.274,Z 452.196,A -85,B 0,C 180,E1 -1732.052,E2 -1732.052} C_VEL
LIN {X 0,Y 580.307,Z 452.201,A -85,B 0,C 180,E1 -1735.079,E2 -1735.079} C_VEL
LIN {X 0,Y 580.3,Z 452.192,A -85,B 0,C 180,E1 -1738.185,E2 -1738.185} C_VEL
LIN {X 0,Y 580.294,Z 452.201,A -85,B 0,C 180,E1 -1740.695,E2 -1740.695} C_VEL
LIN {X 0,Y 580.302,Z 452.2,A -85,B 0,C 180,E1 -1743.316,E2 -1743.316} C_VEL
LIN {X 0,Y 580.268,Z 452.198,A -85,B 0,C 180,E1 -1745.759,E2 -1745.759} C_VEL
LIN {X 0,Y 580.288,Z 452.195,A -85,B 0,C 180,E1 -1748.145,E2 -1748.145} C_VEL
LIN {X 0,Y 580.299,Z 452.201,A -85,B 0,C 180,E1 -1750.842,E2 -1750.842} C_VEL
LIN {X 0,Y 580.285,Z 452.197,A -85,B 0,C 180,E1 -1753.656,E2 -1753.656} C_VEL
LIN {X 0,Y 580.273,Z 452.2,A -85,B 0,C 180,E1 -1756.608,E2 -1756.608} C_VEL
LIN {X 0,Y 580.296,Z 452.201,A -85,B 0,C 180,E1 -1759.156,E2 -1759.156} C_VEL
LIN {X 0,Y 580.285,Z 452.196,A -85,B 0,C 180,E1 -1761.926,E2 -1761.926} C_VEL
LIN {X 0,Y 580.304,Z 452.195,A -85,B 0,C 180,E1 -1764.456,E2 -1764.456} C_VEL
LIN {X 0,Y 580.286,Z 452.202,A -85,B 0,C 180,E1 -1766.975,E2 -1766.975} C_VEL
LIN {X 0,Y 580.303,Z 452.197,A -85,B 0,C 180,E1 -1769.425,E2 -1769.425} C_VEL
LIN {X 0,Y 580.312,Z 452.191,A -85,B 0,C 180,E1 -1772.136,E2 -1772.136} C_VEL
LIN {X 0,Y 580.302,Z 452.199,A -85,B 0,C 180,E1 -1774.92,E2 -1774.92} C_VEL
LIN {X 0,Y 580.267,Z 452.198,A -85,B 0,C 180,E1 -1777.947,E2 -1777.947} C_VEL
LIN {X 0,Y 580.309,Z 452.197,A -85,B 0,C 180,E1 -1780.914,E2 -1780.914} C_VEL
LIN {X 0,Y 580.273,Z 452.199,A -85,B 0,C 180,E1 -1783.825,E2 -1783.825} C_VEL
LIN {X 0,Y 580.316,Z 452.193,A -85,B 0,C 180,E1 -1785.983,E2 -1785.983} C_VEL
LIN {X 0,Y 580.321,Z 452.194,A -85,B 0,C 180,E1 -1788.827,E2 -1788.827} C_VEL
LIN {X 0,Y 580.328,Z 452.196,A -85,B 0,C 180,E1 -1791.644,E2 -1791.644} C_VEL
LIN {X 0,Y 580.317,Z 452.192,A -85,B 0,C 180,E1 -1794.44,E2 -1794.44} C_VEL
LIN {X 0,Y 580.341,Z 452.195,A -85,B 0,C 180,E1 -1797.223,E2 -1797.223} C_VEL
LIN {X 0,Y 580.342,Z 452.191,A -85,B 0,C 180,E1 -1800,E2 -1800} C_VEL
LIN {X 0,Y 580.34,Z 452.189,A -85,B 0,C 180,E1 -1802.777,E2 -1802.777} C_VEL
LIN {X 0,Y 580.318,Z 452.201,A -85,B 0,C 180,E1 -1805.56,E2 -1805.56} C_VEL
LIN {X 0,Y 580.327,Z 452.191,A -85,B 0,C 180,E1 -1808.356,E2 -1808.356} C_VEL
LIN {X 0,Y 580.323,Z 452.195,A -85,B 0,C 180,E1 -1811.209,E2 -1811.209} C_VEL
LIN {X 0,Y 580.305,Z 452.194,A -85,B 0,C 180,E1 -1814.339,E2 -1814.339} C_VEL
LIN {X 0,Y 580.303,Z 452.194,A -85,B 0,C 180,E1 -1816.915,E2 -1816.915} C_VEL
LIN {X 0,Y 580.299,Z 452.2,A -85,B 0,C 180,E1 -1819.823,E2 -1819.823} C_VEL
LIN {X 0,Y 580.266,Z 452.202,A -85,B 0,C 180,E1 -1822.053,E2 -1822.053} C_VEL
LIN {X 0,Y 580.301,Z 452.196,A -85,B 0,C 180,E1 -1825.08,E2 -1825.08} C_VEL
LIN {X 0,Y 580.312,Z 452.199,A -85,B 0,C 180,E1 -1827.864,E2 -1827.864} C_VEL
LIN {X 0,Y 580.291,Z 452.195,A -85,B 0,C 180,E1 -1830.698,E2 -1830.698} C_VEL
LIN {X 0,Y 580.298,Z 452.197,A -85,B 0,C 180,E1 -1833.317,E2 -1833.317} C_VEL
LIN {X 0,Y 580.321,Z 452.201,A -85,B 0,C 180,E1 -1835.768,E2 -1835.768} C_VEL
LIN {X 0,Y 580.283,Z 452.199,A -85,B 0,C 180,E1 -1838.147,E2 -1838.147} C_VEL
LIN {X 0,Y 580.294,Z 452.195,A -85,B 0,C 180,E1 -1840.844,E2 -1840.844} C_VEL
LIN {X 0,Y 580.273,Z 452.204,A -85,B 0,C 180,E1 -1843.659,E2 -1843.659} C_VEL
LIN {X 0,Y 580.282,Z 452.197,A -85,B 0,C 180,E1 -1846.609,E2 -1846.609} C_VEL
LIN {X 0,Y 580.298,Z 452.195,A -85,B 0,C 180,E1 -1849.158,E2 -1849.158} C_VEL
LIN {X 0,Y 580.289,Z 452.204,A -85,B 0,C 180,E1 -1851.927,E2 -1851.927} C_VEL
LIN {X 0,Y 580.278,Z 452.199,A -85,B 0,C 180,E1 -1854.456,E2 -1854.456} C_VEL
LIN {X 0,Y 580.29,Z 452.195,A -85,B 0,C 180,E1 -1856.976,E2 -1856.976} C_VEL
LIN {X 0,Y 580.302,Z 452.197,A -85,B 0,C 180,E1 -1859.426,E2 -1859.426} C_VEL
LIN {X 0,Y 580.299,Z 452.202,A -85,B 0,C 180,E1 -1862.142,E2 -1862.142} C_VEL
LIN {X 0,Y 580.316,Z 452.337,A -85,B 0,C 180,E1 -1862.893,E2 -1862.893} C_VEL
LIN {X 0,Y 581.681,Z 458.082,A -85,B 0,C 180,E1 -1863.629,E2 -1863.629} C_VEL
LIN {X 0,Y 581.444,Z 481.712,A -85,B 0,C 180,E1 -1866.304,E2 -1866.304} C_VEL
LIN {X 0,Y 581.086,Z 508.608,A -85,B 0,C 180,E1 -1869.283,E2 -1869.283} C_VEL
LIN {X 0,Y 580.808,Z 535.503,A -85,B 0,C 180,E1 -1872.21,E2 -1872.21} C_VEL
LIN {X 0,Y 580.62,Z 560.718,A -85,B 0,C 180,E1 -1874.916,E2 -1874.916} C_VEL
LIN {X 0,Y 580.528,Z 573.897,A -85,B 0,C 180,E1 -1876.301,E2 -1876.301} C_VEL
LIN {X 0,Y 580.985,Z 579.746,A -85,B 0,C 180,E1 -1876.401,E2 -1876.401} C_VEL
LIN {X 0,Y 580.83,Z 683.962,A -85,B 0,C 180,E1 -1877.709,E2 -1877.709} C_VEL
LIN {X 0,Y 580.752,Z 696.468,A -85,B 0,C 180,E1 -1877.995,E2 -1877.995} C_VEL
LIN {X 0,Y 580.658,Z 709.379,A -85,B 0,C 180,E1 -1878.436,E2 -1878.436} C_VEL
LIN {X 0,Y 580.564,Z 721.635,A -85,B 0,C 180,E1 -1879.009,E2 -1879.009} C_VEL
LIN {X 0,Y 580.443,Z 733.206,A -85,B 0,C 180,E1 -1879.712,E2 -1879.712} C_VEL
LIN {X 0,Y 580.341,Z 743.601,A -85,B 0,C 180,E1 -1880.503,E2 -1880.503} C_VEL
LIN {X 0,Y 580.271,Z 752.114,A -85,B 0,C 180,E1 -1881.292,E2 -1881.292} C_VEL
LIN {X 0,Y 580.221,Z 759.962,A -85,B 0,C 180,E1 -1882.168,E2 -1882.168} C_VEL
LIN {X 0,Y 580.153,Z 767.651,A -85,B 0,C 180,E1 -1883.222,E2 -1883.222} C_VEL
LIN {X 0,Y 580.139,Z 774.681,A -85,B 0,C 180,E1 -1884.439,E2 -1884.439} C_VEL
LIN {X 0,Y 580.108,Z 779.372,A -85,B 0,C 180,E1 -1885.484,E2 -1885.484} C_VEL
LIN {X 0,Y 580.123,Z 782.957,A -85,B 0,C 180,E1 -1886.527,E2 -1886.527} C_VEL
LIN {X 0,Y 580.043,Z 784.809,A -85,B 0,C 180,E1 -1887.222,E2 -1887.222} C_VEL
LIN {X 0,Y 580.038,Z 786.2,A -85,B 0,C 180,E1 -1887.917,E2 -1887.917} C_VEL
LIN {X 0,Y 580.04,Z 787.784,A -85,B 0,C 180,E1 -1889.306,E2 -1889.306} C_VEL
LIN {X 0,Y 580.037,Z 788,A -85,B 0,C 180,E1 -1890,E2 -1890} C_VEL
LIN {X 0,Y 580.047,Z 787.186,A -85,B 0,C 180,E1 -1891.389,E2 -1891.389} C_VEL
LIN {X 0,Y 580.038,Z 786.201,A -85,B 0,C 180,E1 -1892.083,E2 -1892.083} C_VEL
LIN {X 0,Y 580.043,Z 784.81,A -85,B 0,C 180,E1 -1892.778,E2 -1892.778} C_VEL
LIN {X 0,Y 580.109,Z 781.896,A -85,B 0,C 180,E1 -1893.82,E2 -1893.82} C_VEL
LIN {X 0,Y 580.054,Z 777.95,A -85,B 0,C 180,E1 -1894.865,E2 -1894.865} C_VEL
LIN {X 0,Y 580.139,Z 771.878,A -85,B 0,C 180,E1 -1896.085,E2 -1896.085} C_VEL
LIN {X 0,Y 580.184,Z 765.238,A -85,B 0,C 180,E1 -1897.132,E2 -1897.132} C_VEL
LIN {X 0,Y 580.25,Z 756.992,A -85,B 0,C 180,E1 -1898.182,E2 -1898.182} C_VEL
LIN {X 0,Y 580.308,Z 748.54,A -85,B 0,C 180,E1 -1899.058,E2 -1899.058} C_VEL
LIN {X 0,Y 580.415,Z 738.099,A -85,B 0,C 180,E1 -1899.936,E2 -1899.936} C_VEL
LIN {X 0,Y 580.496,Z 727.761,A -85,B 0,C 180,E1 -1900.639,E2 -1900.639} C_VEL
LIN {X 0,Y 580.597,Z 716.236,A -85,B 0,C 180,E1 -1901.264,E2 -1901.264} C_VEL
LIN {X 0,Y 580.674,Z 703.48,A -85,B 0,C 180,E1 -1901.785,E2 -1901.785} C_VEL
LIN {X 0,Y 580.737,Z 690.447,A -85,B 0,C 180,E1 -1902.16,E2 -1902.16} C_VEL
LIN {X 0,Y 580.831,Z 678.106,A -85,B 0,C 180,E1 -1902.38,E2 -1902.38} C_VEL
LIN {X 0,Y 580.802,Z 576.169,A -85,B 0,C 180,E1 -1903.648,E2 -1903.648} C_VEL
LIN {X 0,Y 580.517,Z 573.578,A -85,B 0,C 180,E1 -1903.722,E2 -1903.722} C_VEL
LIN {X 0,Y 580.739,Z 547.27,A -85,B 0,C 180,E1 -1906.522,E2 -1906.522} C_VEL
LIN {X 0,Y 580.953,Z 519.749,A -85,B 0,C 180,E1 -1909.499,E2 -1909.499} C_VEL
LIN {X 0,Y 581.264,Z 493.479,A -85,B 0,C 180,E1 -1912.387,E2 -1912.387} C_VEL
LIN {X 0,Y 581.583,Z 469.945,A -85,B 0,C 180,E1 -1915.02,E2 -1915.02} C_VEL
LIN {X 0,Y 581.688,Z 458.067,A -85,B 0,C 180,E1 -1916.373,E2 -1916.373} C_VEL
LIN {X 0,Y 580.304,Z 452.266,A -85,B 0,C 180,E1 -1917.132,E2 -1917.132} C_VEL
LIN {X 0,Y 580.287,Z 452.198,A -85,B 0,C 180,E1 -1919.772,E2 -1919.772} C_VEL
LIN {X 0,Y 580.301,Z 452.203,A -85,B 0,C 180,E1 -1922.199,E2 -1922.199} C_VEL
LIN {X 0,Y 580.287,Z 452.199,A -85,B 0,C 180,E1 -1924.695,E2 -1924.695} C_VEL
LIN {X 0,Y 580.297,Z 452.194,A -85,B 0,C 180,E1 -1927.267,E2 -1927.267} C_VEL
LIN {X 0,Y 580.295,Z 452.203,A -85,B 0,C 180,E1 -1930.271,E2 -1930.271} C_VEL
LIN {X 0,Y 580.279,Z 452.2,A -85,B 0,C 180,E1 -1932.705,E2 -1932.705} C_VEL
LIN {X 0,Y 580.265,Z 452.198,A -85,B 0,C 180,E1 -1935.608,E2 -1935.608} C_VEL
LIN {X 0,Y 580.308,Z 452.202,A -85,B 0,C 180,E1 -1938.234,E2 -1938.234} C_VEL
LIN {X 0,Y 580.284,Z 452.196,A -85,B 0,C 180,E1 -1940.965,E2 -1940.965} C_VEL
LIN {X 0,Y 580.29,Z 452.196,A -85,B 0,C 180,E1 -1943.598,E2 -1943.598} C_VEL
LIN {X 0,Y 580.314,Z 452.2,A -85,B 0,C 180,E1 -1946.145,E2 -1946.145} C_VEL
LIN {X 0,Y 580.283,Z 452.202,A -85,B 0,C 180,E1 -1948.615,E2 -1948.615} C_VEL
LIN {X 0,Y 580.289,Z 452.196,A -85,B 0,C 180,E1 -1951.024,E2 -1951.024} C_VEL
LIN {X 0,Y 580.321,Z 452.19,A -85,B 0,C 180,E1 -1953.658,E2 -1953.658} C_VEL
LIN {X 0,Y 580.272,Z 452.208,A -85,B 0,C 180,E1 -1956.442,E2 -1956.442} C_VEL
LIN {X 0,Y 580.274,Z 452.196,A -85,B 0,C 180,E1 -1959.437,E2 -1959.437} C_VEL
LIN {X 0,Y 580.274,Z 452.195,A -85,B 0,C 180,E1 -1961.645,E2 -1961.645} C_VEL
LIN {X 0,Y 580.274,Z 452.198,A -85,B 0,C 180,E1 -1963.825,E2 -1963.825} C_VEL
LIN {X 0,Y 580.316,Z 452.195,A -85,B 0,C 180,E1 -1965.983,E2 -1965.983} C_VEL
LIN {X 0,Y 580.321,Z 452.195,A -85,B 0,C 180,E1 -1968.827,E2 -1968.827} C_VEL
LIN {X 0,Y 580.326,Z 452.191,A -85,B 0,C 180,E1 -1971.644,E2 -1971.644} C_VEL
LIN {X 0,Y 580.319,Z 452.2,A -85,B 0,C 180,E1 -1974.44,E2 -1974.44} C_VEL
LIN {X 0,Y 580.34,Z 452.19,A -85,B 0,C 180,E1 -1977.223,E2 -1977.223} C_VEL
LIN {X 0,Y 580.342,Z 452.191,A -85,B 0,C 180,E1 -1980,E2 -1980} C_VEL
LIN {X 0,Y 580.341,Z 452.196,A -85,B 0,C 180,E1 -1982.777,E2 -1982.777} C_VEL
LIN {X 0,Y 580.322,Z 452.191,A -85,B 0,C 180,E1 -1985.56,E2 -1985.56} C_VEL
LIN {X 0,Y 580.328,Z 452.195,A -85,B 0,C 180,E1 -1988.356,E2 -1988.356} C_VEL
LIN {X 0,Y 580.323,Z 452.193,A -85,B 0,C 180,E1 -1991.209,E2 -1991.209} C_VEL
LIN {X 0,Y 580.305,Z 452.198,A -85,B 0,C 180,E1 -1994.339,E2 -1994.339} C_VEL
LIN {X 0,Y 580.304,Z 452.201,A -85,B 0,C 180,E1 -1996.915,E2 -1996.915} C_VEL
LIN {X 0,Y 580.3,Z 452.194,A -85,B 0,C 180,E1 -1999.823,E2 -1999.823} C_VEL
LIN {X 0,Y 580.278,Z 452.198,A -85,B 0,C 180,E1 -2001.347,E2 -2001.347} C_VEL
LIN {X 0,Y 579.581,Z 452.285,A -85,B 0,C 180,E1 -2001.926,E2 -2001.926} C_VEL
LIN {X 0,Y 576.704,Z 452.651,A -85,B 0,C 180,E1 -2002.866,E2 -2002.866} C_VEL
LIN {X 0,Y 574.309,Z 452.944,A -85,B 0,C 180,E1 -2003.622,E2 -2003.622} C_VEL
LIN {X 0,Y 573.31,Z 453.067,A -85,B 0,C 180,E1 -2004.206,E2 -2004.206} C_VEL
LIN {X 0,Y 573.244,Z 453.077,A -85,B 0,C 180,E1 -2004.403,E2 -2004.403} C_VEL
LIN {X 0,Y 573.257,Z 453.078,A -85,B 0,C 180,E1 -2006.976,E2 -2006.976} C_VEL
LIN {X 0,Y 573.247,Z 453.069,A -85,B 0,C 180,E1 -2009.491,E2 -2009.491} C_VEL
LIN {X 0,Y 573.249,Z 453.07,A -85,B 0,C 180,E1 -2012.23,E2 -2012.23} C_VEL
LIN {X 0,Y 573.249,Z 453.081,A -85,B 0,C 180,E1 -2014.775,E2 -2014.775} C_VEL
LIN {X 0,Y 573.249,Z 453.077,A -85,B 0,C 180,E1 -2017.167,E2 -2017.167} C_VEL
LIN {X 0,Y 573.244,Z 453.069,A -85,B 0,C 180,E1 -2019.608,E2 -2019.608} C_VEL
LIN {X 0,Y 573.239,Z 453.078,A -85,B 0,C 180,E1 -2022.643,E2 -2022.643} C_VEL
LIN {X 0,Y 573.236,Z 453.074,A -85,B 0,C 180,E1 -2025.668,E2 -2025.668} C_VEL
LIN {X 0,Y 573.243,Z 453.074,A -85,B 0,C 180,E1 -2028.545,E2 -2028.545} C_VEL
LIN {X 0,Y 573.249,Z 453.077,A -85,B 0,C 180,E1 -2031.3,E2 -2031.3} C_VEL
LIN {X 0,Y 573.242,Z 453.069,A -85,B 0,C 180,E1 -2034.015,E2 -2034.015} C_VEL
LIN {X 0,Y 573.285,Z 453.064,A -85,B 0,C 180,E1 -2036.52,E2 -2036.52} C_VEL
LIN {X 0,Y 573.24,Z 453.084,A -85,B 0,C 180,E1 -2039.117,E2 -2039.117} C_VEL
LIN {X 0,Y 573.252,Z 453.07,A -85,B 0,C 180,E1 -2041.972,E2 -2041.972} C_VEL
LIN {X 0,Y 573.255,Z 453.073,A -85,B 0,C 180,E1 -2044.591,E2 -2044.591} C_VEL
LIN {X 0,Y 573.239,Z 453.075,A -85,B 0,C 180,E1 -2047.663,E2 -2047.663} C_VEL
LIN {X 0,Y 573.281,Z 453.073,A -85,B 0,C 180,E1 -2050.729,E2 -2050.729} C_VEL
LIN {X 0,Y 573.254,Z 453.073,A -85,B 0,C 180,E1 -2053.622,E2 -2053.622} C_VEL
LIN {X 0,Y 573.308,Z 453.198,A -85,B 0,C 180,E1 -2056.441,E2 -2056.441} C_VEL
LIN {X 0,Y 573.508,Z 454.132,A -85,B 0,C 180,E1 -2056.559,E2 -2056.559} C_VEL
LIN {X 0,Y 574.04,Z 456.578,A -85,B 0,C 180,E1 -2056.617,E2 -2056.617} C_VEL
LIN {X 0,Y 573.911,Z 533.96,A -85,B 0,C 180,E1 -2057.603,E2 -2057.603} C_VEL
LIN {X 0,Y 573.815,Z 547.227,A -85,B 0,C 180,E1 -2057.915,E2 -2057.915} C_VEL
LIN {X 0,Y 573.717,Z 559.384,A -85,B 0,C 180,E1 -2058.339,E2 -2058.339} C_VEL
LIN {X 0,Y 573.611,Z 570.864,A -85,B 0,C 180,E1 -2058.877,E2 -2058.877} C_VEL
LIN {X 0,Y 573.442,Z 582.552,A -85,B 0,C 180,E1 -2059.585,E2 -2059.585} C_VEL
LIN {X 0,Y 573.331,Z 593.07,A -85,B 0,C 180,E1 -2060.386,E2 -2060.386} C_VEL
LIN {X 0,Y 573.241,Z 601.667,A -85,B 0,C 180,E1 -2061.185,E2 -2061.185} C_VEL
LIN {X 0,Y 573.161,Z 609.588,A -85,B 0,C 180,E1 -2062.071,E2 -2062.071} C_VEL
LIN {X 0,Y 573.093,Z 617.524,A -85,B 0,C 180,E1 -2063.163,E2 -2063.163} C_VEL
LIN {X 0,Y 573.07,Z 624.45,A -85,B 0,C 180,E1 -2064.37,E2 -2064.37} C_VEL
LIN {X 0,Y 573.028,Z 629.192,A -85,B 0,C 180,E1 -2065.428,E2 -2065.428} C_VEL
LIN {X 0,Y 573.022,Z 632.825,A -85,B 0,C 180,E1 -2066.484,E2 -2066.484} C_VEL
LIN {X 0,Y 572.959,Z 634.702,A -85,B 0,C 180,E1 -2067.188,E2 -2067.188} C_VEL
LIN {X 0,Y 572.939,Z 636.127,A -85,B 0,C 180,E1 -2067.891,E2 -2067.891} C_VEL
LIN {X 0,Y 572.941,Z 637.756,A -85,B 0,C 180,E1 -2069.297,E2 -2069.297} C_VEL
LIN {X 0,Y 572.939,Z 637.996,A -85,B 0,C 180,E1 -2070,E2 -2070} C_VEL
LIN {X 0,Y 572.94,Z 637.815,A -85,B 0,C 180,E1 -2070.703,E2 -2070.703} C_VEL
LIN {X 0,Y 572.939,Z 636.271,A -85,B 0,C 180,E1 -2072.109,E2 -2072.109} C_VEL
LIN {X 0,Y 572.96,Z 634.91,A -85,B 0,C 180,E1 -2072.812,E2 -2072.812} C_VEL
LIN {X 0,Y 573.015,Z 632.031,A -85,B 0,C 180,E1 -2073.868,E2 -2073.868} C_VEL
LIN {X 0,Y 572.963,Z 628.132,A -85,B 0,C 180,E1 -2074.926,E2 -2074.926} C_VEL
LIN {X 0,Y 573.075,Z 623.1,A -85,B 0,C 180,E1 -2075.983,E2 -2075.983} C_VEL
LIN {X 0,Y 573.083,Z 616.777,A -85,B 0,C 180,E1 -2077.044,E2 -2077.044} C_VEL
LIN {X 0,Y 573.178,Z 608.855,A -85,B 0,C 180,E1 -2078.106,E2 -2078.106} C_VEL
LIN {X 0,Y 573.287,Z 599.005,A -85,B 0,C 180,E1 -2079.17,E2 -2079.17} C_VEL
LIN {X 0,Y 573.423,Z 588.692,A -85,B 0,C 180,E1 -2080.058,E2 -2080.058} C_VEL
LIN {X 0,Y 573.562,Z 577.107,A -85,B 0,C 180,E1 -2080.855,E2 -2080.855} C_VEL
LIN {X 0,Y 573.643,Z 565.498,A -85,B 0,C 180,E1 -2081.483,E2 -2081.483} C_VEL
LIN {X 0,Y 573.758,Z 553.494,A -85,B 0,C 180,E1 -2081.974,E2 -2081.974} C_VEL
LIN {X 0,Y 573.85,Z 540.458,A -85,B 0,C 180,E1 -2082.353,E2 -2082.353} C_VEL
LIN {X 0,Y 573.943,Z 528.114,A -85,B 0,C 180,E1 -2082.576,E2 -2082.576} C_VEL
LIN {X 0,Y 573.896,Z 455.562,A -85,B 0,C 180,E1 -2083.49,E2 -2083.49} C_VEL
LIN {X 0,Y 573.408,Z 453.794,A -85,B 0,C 180,E1 -2083.556,E2 -2083.556} C_VEL
LIN {X 0,Y 573.295,Z 453.107,A -85,B 0,C 180,E1 -2083.695,E2 -2083.695} C_VEL
LIN {X 0,Y 573.262,Z 453.067,A -85,B 0,C 180,E1 -2087.009,E2 -2087.009} C_VEL
LIN {X 0,Y 573.254,Z 453.073,A -85,B 0,C 180,E1 -2090.076,E2 -2090.076} C_VEL
LIN {X 0,Y 573.236,Z 453.082,A -85,B 0,C 180,E1 -2093.099,E2 -2093.099} C_VEL
LIN {X 0,Y 573.254,Z 453.074,A -85,B 0,C 180,E1 -2095.409,E2 -2095.409} C_VEL
LIN {X 0,Y 573.252,Z 453.069,A -85,B 0,C 180,E1 -2098.028,E2 -2098.028} C_VEL
LIN {X 0,Y 573.24,Z 453.083,A -85,B 0,C 180,E1 -2100.883,E2 -2100.883} C_VEL
LIN {X 0,Y 573.261,Z 453.074,A -85,B 0,C 180,E1 -2103.523,E2 -2103.523} C_VEL
LIN {X 0,Y 573.241,Z 453.073,A -85,B 0,C 180,E1 -2106.049,E2 -2106.049} C_VEL
LIN {X 0,Y 573.248,Z 453.077,A -85,B 0,C 180,E1 -2108.7,E2 -2108.7} C_VEL
LIN {X 0,Y 573.251,Z 453.073,A -85,B 0,C 180,E1 -2111.595,E2 -2111.595} C_VEL
LIN {X 0,Y 573.235,Z 453.074,A -85,B 0,C 180,E1 -2114.332,E2 -2114.332} C_VEL
LIN {X 0,Y 573.236,Z 453.08,A -85,B 0,C 180,E1 -2117.358,E2 -2117.358} C_VEL
LIN {X 0,Y 573.244,Z 453.069,A -85,B 0,C 180,E1 -2120.392,E2 -2120.392} C_VEL
LIN {X 0,Y 573.251,Z 453.08,A -85,B 0,C 180,E1 -2123.077,E2 -2123.077} C_VEL
LIN {X 0,Y 573.27,Z 453.072,A -85,B 0,C 180,E1 -2125.671,E2 -2125.671} C_VEL
LIN {X 0,Y 573.243,Z 453.069,A -85,B 0,C 180,E1 -2128.184,E2 -2128.184} C_VEL
LIN {X 0,Y 573.264,Z 453.068,A -85,B 0,C 180,E1 -2130.634,E2 -2130.634} C_VEL
LIN {X 0,Y 573.263,Z 453.077,A -85,B 0,C 180,E1 -2133.5,E2 -2133.5} C_VEL
LIN {X 0,Y 573.225,Z 453.075,A -85,B 0,C 180,E1 -2136.134,E2 -2136.134} C_VEL
LIN {X 0,Y 573.253,Z 453.079,A -85,B 0,C 180,E1 -2139.174,E2 -2139.174} C_VEL
LIN {X 0,Y 573.231,Z 453.083,A -85,B 0,C 180,E1 -2141.411,E2 -2141.411} C_VEL
LIN {X 0,Y 573.249,Z 453.076,A -85,B 0,C 180,E1 -2143.622,E2 -2143.622} C_VEL
LIN {X 0,Y 573.228,Z 453.075,A -85,B 0,C 180,E1 -2146.529,E2 -2146.529} C_VEL
LIN {X 0,Y 573.273,Z 453.071,A -85,B 0,C 180,E1 -2148.734,E2 -2148.734} C_VEL
LIN {X 0,Y 573.299,Z 453.073,A -85,B 0,C 180,E1 -2151.541,E2 -2151.541} C_VEL
LIN {X 0,Y 573.284,Z 453.068,A -85,B 0,C 180,E1 -2154.372,E2 -2154.372} C_VEL
LIN {X 0,Y 573.3,Z 453.068,A -85,B 0,C 180,E1 -2157.892,E2 -2157.892} C_VEL
LIN {X 0,Y 573.329,Z 453.063,A -85,B 0,C 180,E1 -2160.702,E2 -2160.702} C_VEL
LIN {X 0,Y 573.234,Z 453.082,A -85,B 0,C 180,E1 -2163.514,E2 -2163.514} C_VEL
LIN {X 0,Y 573.285,Z 453.076,A -85,B 0,C 180,E1 -2165.628,E2 -2165.628} C_VEL
LIN {X 0,Y 573.298,Z 453.066,A -85,B 0,C 180,E1 -2168.459,E2 -2168.459} C_VEL
LIN {X 0,Y 573.289,Z 453.072,A -85,B 0,C 180,E1 -2171.312,E2 -2171.312} C_VEL
LIN {X 0,Y 573.271,Z 453.07,A -85,B 0,C 180,E1 -2174.425,E2 -2174.425} C_VEL
LIN {X 0,Y 573.25,Z 453.074,A -85,B 0,C 180,E1 -2177.112,E2 -2177.112} C_VEL
LIN {X 0,Y 573.248,Z 453.074,A -85,B 0,C 180,E1 -2180.077,E2 -2180.077} C_VEL
LIN {X 0,Y 573.229,Z 453.076,A -85,B 0,C 180,E1 -2182.338,E2 -2182.338} C_VEL
LIN {X 0,Y 573.25,Z 453.079,A -85,B 0,C 180,E1 -2185.41,E2 -2185.41} C_VEL
LIN {X 0,Y 573.256,Z 453.075,A -85,B 0,C 180,E1 -2188.032,E2 -2188.032} C_VEL
LIN {X 0,Y 573.236,Z 453.075,A -85,B 0,C 180,E1 -2190.886,E2 -2190.886} C_VEL
LIN {X 0,Y 573.281,Z 453.074,A -85,B 0,C 180,E1 -2193.529,E2 -2193.529} C_VEL
LIN {X 0,Y 573.255,Z 453.077,A -85,B 0,C 180,E1 -2196.049,E2 -2196.049} C_VEL
LIN {X 0,Y 573.243,Z 453.072,A -85,B 0,C 180,E1 -2198.702,E2 -2198.702} C_VEL
LIN {X 0,Y 573.248,Z 453.081,A -85,B 0,C 180,E1 -2201.596,E2 -2201.596} C_VEL
LIN {X 0,Y 573.23,Z 453.075,A -85,B 0,C 180,E1 -2204.334,E2 -2204.334} C_VEL
LIN {X 0,Y 573.24,Z 453.078,A -85,B 0,C 180,E1 -2207.359,E2 -2207.359} C_VEL
LIN {X 0,Y 573.245,Z 453.075,A -85,B 0,C 180,E1 -2210.394,E2 -2210.394} C_VEL
LIN {X 0,Y 573.252,Z 453.072,A -85,B 0,C 180,E1 -2213.079,E2 -2213.079} C_VEL
LIN {X 0,Y 573.265,Z 453.079,A -85,B 0,C 180,E1 -2215.672,E2 -2215.672} C_VEL
LIN {X 0,Y 573.248,Z 453.078,A -85,B 0,C 180,E1 -2218.186,E2 -2218.186} C_VEL
LIN {X 0,Y 573.263,Z 453.074,A -85,B 0,C 180,E1 -2220.635,E2 -2220.635} C_VEL
LIN {X 0,Y 573.276,Z 453.235,A -85,B 0,C 180,E1 -2222.73,E2 -2222.73} C_VEL
LIN {X 0,Y 574.882,Z 460.296,A -85,B 0,C 180,E1 -2223.592,E2 -2223.592} C_VEL
LIN {X 0,Y 574.631,Z 480.031,A -85,B 0,C 180,E1 -2225.813,E2 -2225.813} C_VEL
LIN {X 0,Y 574.317,Z 503.565,A -85,B 0,C 180,E1 -2228.463,E2 -2228.463} C_VEL
LIN {X 0,Y 573.96,Z 530.46,A -85,B 0,C 180,E1 -2231.436,E2 -2231.436} C_VEL
LIN {X 0,Y 573.677,Z 555.675,A -85,B 0,C 180,E1 -2234.183,E2 -2234.183} C_VEL
LIN {X 0,Y 573.555,Z 573.896,A -85,B 0,C 180,E1 -2236.131,E2 -2236.131} C_VEL
LIN {X 0,Y 574.091,Z 579.746,A -85,B 0,C 180,E1 -2236.235,E2 -2236.235} C_VEL
LIN {X 0,Y 573.908,Z 683.962,A -85,B 0,C 180,E1 -2237.558,E2 -2237.558} C_VEL
LIN {X 0,Y 573.825,Z 696.467,A -85,B 0,C 180,E1 -2237.848,E2 -2237.848} C_VEL
LIN {X 0,Y 573.703,Z 708.924,A -85,B 0,C 180,E1 -2238.276,E2 -2238.276} C_VEL
LIN {X 0,Y 573.595,Z 720.443,A -85,B 0,C 180,E1 -2238.81,E2 -2238.81} C_VEL
LIN {X 0,Y 573.471,Z 731.915,A -85,B 0,C 180,E1 -2239.497,E2 -2239.497} C_VEL
LIN {X 0,Y 573.343,Z 742.543,A -85,B 0,C 180,E1 -2240.297,E2 -2240.297} C_VEL
LIN {X 0,Y 573.241,Z 752.115,A -85,B 0,C 180,E1 -2241.185,E2 -2241.185} C_VEL
LIN {X 0,Y 573.161,Z 759.962,A -85,B 0,C 180,E1 -2242.071,E2 -2242.071} C_VEL
LIN {X 0,Y 573.072,Z 767.955,A -85,B 0,C 180,E1 -2243.186,E2 -2243.186} C_VEL
LIN {X 0,Y 573.07,Z 774.681,A -85,B 0,C 180,E1 -2244.37,E2 -2244.37} C_VEL
LIN {X 0,Y 573.029,Z 779.372,A -85,B 0,C 180,E1 -2245.428,E2 -2245.428} C_VEL
LIN {X 0,Y 573.022,Z 782.957,A -85,B 0,C 180,E1 -2246.484,E2 -2246.484} C_VEL
LIN {X 0,Y 572.959,Z 784.808,A -85,B 0,C 180,E1 -2247.188,E2 -2247.188} C_VEL
LIN {X 0,Y 572.937,Z 786.199,A -85,B 0,C 180,E1 -2247.891,E2 -2247.891} C_VEL
LIN {X 0,Y 572.941,Z 787.785,A -85,B 0,C 180,E1 -2249.297,E2 -2249.297} C_VEL
LIN {X 0,Y 572.938,Z 788,A -85,B 0,C 180,E1 -2250,E2 -2250} C_VEL
LIN {X 0,Y 572.946,Z 787.186,A -85,B 0,C 180,E1 -2251.406,E2 -2251.406} C_VEL
LIN {X 0,Y 572.937,Z 786.2,A -85,B 0,C 180,E1 -2252.109,E2 -2252.109} C_VEL
LIN {X 0,Y 572.959,Z 784.81,A -85,B 0,C 180,E1 -2252.812,E2 -2252.812} C_VEL
LIN {X 0,Y 573.014,Z 781.896,A -85,B 0,C 180,E1 -2253.868,E2 -2253.868} C_VEL
LIN {X 0,Y 572.963,Z 777.95,A -85,B 0,C 180,E1 -2254.925,E2 -2254.925} C_VEL
LIN {X 0,Y 573.064,Z 771.878,A -85,B 0,C 180,E1 -2256.16,E2 -2256.16} C_VEL
LIN {X 0,Y 573.119,Z 765.239,A -85,B 0,C 180,E1 -2257.221,E2 -2257.221} C_VEL
LIN {X 0,Y 573.201,Z 756.992,A -85,B 0,C 180,E1 -2258.283,E2 -2258.283} C_VEL
LIN {X 0,Y 573.286,Z 748.541,A -85,B 0,C 180,E1 -2259.17,E2 -2259.17} C_VEL
LIN {X 0,Y 573.409,Z 738.1,A -85,B 0,C 180,E1 -2260.058,E2 -2260.058} C_VEL
LIN {X 0,Y 573.55,Z 726.356,A -85,B 0,C 180,E1 -2260.857,E2 -2260.857} C_VEL
LIN {X 0,Y 573.652,Z 715.287,A -85,B 0,C 180,E1 -2261.447,E2 -2261.447} C_VEL
LIN {X 0,Y 573.758,Z 702.182,A -85,B 0,C 180,E1 -2261.974,E2 -2261.974} C_VEL
LIN {X 0,Y 573.832,Z 689.532,A -85,B 0,C 180,E1 -2262.331,E2 -2262.331} C_VEL
LIN {X 0,Y 573.898,Z 676.334,A -85,B 0,C 180,E1 -2262.554,E2 -2262.554} C_VEL
LIN {X 0,Y 573.986,Z 577.399,A -85,B 0,C 180,E1 -2263.798,E2 -2263.798} C_VEL
